C09082=1012.478,318.787,350.070,169.822,52.836,160.283
C09083=1012.472,318.539,350.102,169.815,52.841,160.283
C09084=1012.466,318.291,350.134,169.808,52.848,160.283
C09085=1012.460,318.044,350.167,169.801,52.853,160.283
C09086=1012.455,317.796,350.200,169.794,52.859,160.283
C09087=1012.449,317.549,350.233,169.787,52.865,160.283
C09088=1012.443,317.301,350.265,169.780,52.871,160.283
C09089=1012.436,317.053,350.298,169.774,52.876,160.283
C09090=1012.430,316.805,350.330,169.767,52.883,160.283
C09091=1012.424,316.557,350.362,169.760,52.889,160.283
C09092=1012.419,316.309,350.396,169.753,52.894,160.283
C09093=1012.412,316.062,350.429,169.746,52.900,160.283
C09094=1012.406,315.813,350.461,169.739,52.906,160.283
C09095=1012.400,315.566,350.493,169.732,52.912,160.283
C09096=1012.394,315.319,350.526,169.726,52.918,160.283
C09097=1012.388,315.071,350.558,169.719,52.924,160.283
C09098=1012.383,314.823,350.591,169.713,52.929,160.283
C09099=1012.377,314.575,350.623,169.705,52.936,160.283
C09100=1012.370,314.327,350.656,169.699,52.941,160.283
C09101=1012.365,314.080,350.687,169.692,52.948,160.283
C09102=1012.359,313.832,350.720,169.686,52.953,160.283
C09103=1012.353,313.583,350.753,169.678,52.959,160.283
C09104=1012.347,313.336,350.786,169.672,52.965,160.283
C09105=1012.342,313.088,350.817,169.665,52.971,160.283
C09106=1012.336,312.841,350.850,169.659,52.977,160.283
C09107=1012.330,312.593,350.882,169.652,52.983,160.283
C09108=1012.324,312.345,350.914,169.645,52.989,160.283
C09109=1012.319,312.097,350.947,169.638,52.995,160.283
C09110=1012.313,311.849,350.979,169.632,53.001,160.283
C09111=1012.307,311.602,351.011,169.625,53.007,160.283
C09112=1012.301,311.354,351.043,169.618,53.013,160.283
C09113=1012.295,311.106,351.075,169.611,53.019,160.283
C09114=1012.290,310.858,351.107,169.605,53.025,160.283
C09115=1012.284,310.610,351.140,169.598,53.032,160.283
C09116=1012.279,310.363,351.172,169.592,53.037,160.283
C09117=1012.273,310.114,351.204,169.585,53.044,160.283
C09118=1012.267,309.867,351.236,169.579,53.049,160.283
C09119=1012.261,309.619,351.269,169.572,53.056,160.283
C09120=1012.256,309.372,351.300,169.566,53.062,160.284
C09121=1012.250,309.123,351.333,169.558,53.068,160.283
C09122=1012.245,308.876,351.364,169.552,53.074,160.284
C09123=1012.237,308.577,351.403,169.544,53.082,160.284
C09124=1012.230,308.277,351.440,169.536,53.089,160.284
C09125=1012.222,307.977,351.479,169.528,53.097,160.284
C09126=1012.216,307.678,351.516,169.520,53.105,160.284
C09127=1012.209,307.431,351.548,169.514,53.111,160.284
C09128=1012.203,307.182,351.580,169.507,53.118,160.284
C09129=1012.198,306.935,351.610,169.500,53.124,160.284
C09130=1012.192,306.686,351.642,169.494,53.130,160.285
C09131=1012.186,306.439,351.673,169.487,53.136,160.285
C09132=1012.180,306.190,351.704,169.481,53.143,160.285
C09133=1012.174,305.943,351.735,169.474,53.149,160.285
C09134=1012.168,305.695,351.767,169.468,53.155,160.285
C09135=1012.162,305.447,351.798,169.461,53.162,160.285
C09136=1012.156,305.199,351.830,169.454,53.169,160.285
C09137=1012.150,304.951,351.860,169.448,53.175,160.286
C09138=1012.144,304.703,351.892,169.441,53.181,160.285
C09139=1012.138,304.455,351.923,169.435,53.188,160.286
C09140=1012.133,304.207,351.954,169.429,53.195,160.286
C09141=1012.127,303.959,351.985,169.422,53.200,160.286
C09142=1012.121,303.711,352.017,169.416,53.207,160.286
C09143=1012.115,303.464,352.047,169.410,53.214,160.287
C09144=1012.109,303.215,352.079,169.403,53.220,160.287
C09145=1012.104,302.968,352.109,169.396,53.227,160.287
C09146=1012.098,302.719,352.140,169.390,53.233,160.287
C09147=1012.092,302.471,352.172,169.384,53.240,160.287
C09148=1012.087,302.223,352.203,169.378,53.247,160.287
C09149=1012.082,301.975,352.234,169.371,53.253,160.287
C09150=1012.075,301.728,352.265,169.365,53.259,160.288
C09151=1012.070,301.479,352.296,169.358,53.266,160.288
C09152=1012.064,301.231,352.326,169.352,53.273,160.288
C09153=1012.059,300.984,352.358,169.346,53.279,160.288
C09154=1012.053,300.736,352.388,169.339,53.285,160.288
C09155=1012.047,300.487,352.420,169.333,53.292,160.289
C09156=1012.041,300.239,352.450,169.326,53.299,160.289
C09157=1012.036,299.992,352.482,169.320,53.305,160.289
C09158=1012.030,299.744,352.512,169.313,53.312,160.289
C09159=1012.025,299.496,352.543,169.308,53.319,160.289
C09160=1012.019,299.247,352.574,169.301,53.326,160.290
C09161=1012.013,298.999,352.605,169.295,53.332,160.290
C09162=1012.008,298.752,352.635,169.288,53.339,160.290
C09163=1012.002,298.504,352.667,169.283,53.346,160.290
C09164=1011.996,298.256,352.697,169.276,53.352,160.291
C09165=1011.991,298.008,352.728,169.270,53.359,160.291
C09166=1011.986,297.760,352.758,169.263,53.365,160.291
C09167=1011.980,297.512,352.789,169.257,53.373,160.291
C09168=1011.975,297.264,352.820,169.251,53.379,160.291
C09169=1011.969,297.015,352.851,169.244,53.386,160.292
C09170=1011.963,296.768,352.881,169.239,53.393,160.292
C09171=1011.958,296.519,352.912,169.232,53.400,160.292
C09172=1011.952,296.272,352.942,169.226,53.406,160.292
C09173=1011.947,296.024,352.973,169.219,53.413,160.293
C09174=1011.941,295.776,353.004,169.214,53.419,160.293
C09175=1011.936,295.528,353.035,169.207,53.426,160.293
C09176=1011.931,295.279,353.064,169.201,53.433,160.293
C09177=1011.926,295.031,353.095,169.194,53.440,160.293
C09178=1011.920,294.783,353.126,169.189,53.446,160.294
C09179=1011.914,294.503,353.161,169.181,53.454,160.294
C09180=1011.908,294.222,353.195,169.174,53.462,160.294
C09181=1011.903,293.941,353.229,169.168,53.470,160.295
C09182=1011.896,293.661,353.264,169.161,53.478,160.295
C09183=1011.891,293.412,353.294,169.155,53.484,160.295
C09184=1011.885,293.163,353.326,169.148,53.491,160.295
C09185=1011.880,292.915,353.355,169.142,53.499,160.296
C09186=1011.875,292.667,353.386,169.136,53.505,160.296
C09187=1011.870,292.418,353.416,169.129,53.512,160.296
C09188=1011.864,292.170,353.447,169.124,53.519,160.297
C09189=1011.858,291.922,353.477,169.117,53.526,160.297
C09190=1011.853,291.674,353.507,169.112,53.533,160.297
C09191=1011.848,291.427,353.537,169.105,53.540,160.298
C09192=1011.843,291.178,353.567,169.100,53.547,160.298
C09193=1011.837,290.929,353.597,169.093,53.554,160.298
C09194=1011.832,290.682,353.627,169.087,53.561,160.298
C09195=1011.826,290.433,353.657,169.081,53.568,160.299
C09196=1011.820,290.185,353.687,169.075,53.576,160.299
C09197=1011.815,289.938,353.716,169.069,53.582,160.299
C09198=1011.810,289.689,353.746,169.063,53.590,160.300
C09199=1011.804,289.441,353.776,169.057,53.596,160.300
C09200=1011.799,289.193,353.806,169.051,53.604,160.300
C09201=1011.793,288.944,353.835,169.044,53.611,160.301
C09202=1011.788,288.697,353.865,169.039,53.618,160.301
C09203=1011.782,288.449,353.895,169.032,53.625,160.301
C09204=1011.777,288.200,353.925,169.027,53.632,160.302
C09205=1011.771,287.952,353.954,169.021,53.640,160.302
C09206=1011.766,287.704,353.984,169.014,53.647,160.302
C09207=1011.761,287.456,354.013,169.009,53.654,160.303
C09208=1011.755,287.207,354.043,169.002,53.661,160.303
C09209=1011.750,286.960,354.073,168.997,53.668,160.304
C09210=1011.745,286.712,354.102,168.990,53.676,160.304
C09211=1011.739,286.463,354.132,168.984,53.683,160.304
C09212=1011.734,286.216,354.161,168.978,53.690,160.305
C09213=1011.729,285.967,354.191,168.972,53.698,160.305
C09214=1011.723,285.719,354.221,168.967,53.704,160.305
C09215=1011.718,285.471,354.250,168.960,53.712,160.306
C09216=1011.713,285.223,354.280,168.954,53.719,160.306
C09217=1011.707,284.974,354.309,168.949,53.727,160.307
C09218=1011.702,284.726,354.338,168.942,53.734,160.307
C09219=1011.697,284.460,354.369,168.936,53.742,160.307
C09220=1011.691,284.195,354.401,168.930,53.750,160.308
C09221=1011.685,283.929,354.432,168.924,53.757,160.308
C09222=1011.679,283.664,354.464,168.917,53.765,160.308
C09223=1011.451,285.193,353.918,168.925,53.799,160.318
C09224=1011.460,285.578,353.873,168.935,53.789,160.318
C09225=1011.468,285.963,353.827,168.945,53.777,160.317
C09226=1011.477,286.348,353.782,168.954,53.766,160.316
C09227=1011.484,286.732,353.736,168.962,53.754,160.316
C09228=1011.490,286.981,353.706,168.969,53.747,160.316
C09229=1011.495,287.229,353.677,168.975,53.740,160.315
C09230=1011.500,287.477,353.648,168.981,53.733,160.315
C09231=1011.506,287.725,353.618,168.987,53.726,160.315
C09232=1011.511,287.973,353.589,168.992,53.718,160.314
C09233=1011.516,288.221,353.558,168.999,53.711,160.314
C09234=1011.522,288.469,353.529,169.005,53.704,160.314
C09235=1011.527,288.718,353.499,169.011,53.697,160.313
C09236=1011.532,288.966,353.470,169.017,53.690,160.313
C09237=1011.538,289.214,353.440,169.024,53.682,160.313
C09238=1011.544,289.462,353.410,169.029,53.675,160.312
C09239=1011.549,289.710,353.380,169.036,53.668,160.312
C09240=1011.554,289.958,353.351,169.041,53.661,160.312
C09241=1011.560,290.207,353.321,169.048,53.654,160.311
C09242=1011.565,290.454,353.291,169.054,53.647,160.311
C09243=1011.570,290.703,353.261,169.060,53.640,160.311
C09244=1011.575,290.951,353.231,169.066,53.633,160.310
C09245=1011.581,291.199,353.201,169.072,53.626,160.310
C09246=1011.586,291.447,353.171,169.078,53.618,160.310
C09247=1011.592,291.695,353.141,169.085,53.611,160.310
C09248=1011.598,291.943,353.111,169.091,53.605,160.309
C09249=1011.603,292.190,353.081,169.097,53.597,160.309
C09250=1011.608,292.439,353.051,169.103,53.591,160.309
C09251=1011.614,292.687,353.021,169.109,53.584,160.308
C09252=1011.619,292.970,352.986,169.117,53.576,160.308
C09253=1011.625,293.254,352.952,169.123,53.568,160.308
C09254=1011.631,293.539,352.916,169.130,53.560,160.307
C09255=1011.638,293.822,352.882,169.137,53.552,160.307
C09256=1011.643,294.070,352.851,169.143,53.546,160.307
C09257=1011.648,294.317,352.822,169.150,53.539,160.307
C09258=1011.653,294.566,352.791,169.156,53.531,160.306
C09259=1011.659,294.813,352.760,169.162,53.525,160.306
C09260=1011.664,295.062,352.729,169.169,53.518,160.306
C09261=1011.670,295.309,352.699,169.174,53.511,160.306
C09262=1011.675,295.558,352.668,169.181,53.504,160.305
C09263=1011.679,295.806,352.638,169.187,53.498,160.305
C09264=1011.685,296.054,352.607,169.193,53.491,160.305
C09265=1011.690,296.302,352.577,169.199,53.484,160.305
C09266=1011.696,296.550,352.546,169.205,53.477,160.304
C09267=1011.701,296.798,352.515,169.212,53.470,160.304
C09268=1011.707,297.046,352.485,169.218,53.463,160.304
C09269=1011.712,297.294,352.454,169.225,53.457,160.304
C09270=1011.718,297.542,352.424,169.230,53.450,160.303
C09271=1011.723,297.790,352.393,169.237,53.443,160.303
C09272=1011.729,298.038,352.362,169.243,53.437,160.303
C09273=1011.734,298.286,352.331,169.249,53.430,160.303
C09274=1011.740,298.534,352.301,169.255,53.423,160.302
C09275=1011.745,298.782,352.270,169.262,53.416,160.302
C09276=1011.751,299.031,352.239,169.269,53.409,160.302
C09277=1011.756,299.279,352.208,169.275,53.404,160.302
C09278=1011.762,299.526,352.178,169.282,53.397,160.302
C09279=1011.767,299.775,352.147,169.287,53.390,160.302
C09280=1011.773,300.022,352.116,169.294,53.383,160.301
C09281=1011.778,300.270,352.085,169.300,53.377,160.301
C09282=1011.784,300.518,352.055,169.307,53.370,160.301
C09283=1011.790,300.767,352.023,169.313,53.363,160.301
C09284=1011.796,301.014,351.993,169.319,53.356,160.301
C09285=1011.801,301.262,351.961,169.326,53.350,160.301
C09286=1011.807,301.510,351.931,169.332,53.344,160.300
C09287=1011.812,301.758,351.900,169.339,53.337,160.300
C09288=1011.818,302.006,351.869,169.344,53.330,160.300
C09289=1011.824,302.254,351.838,169.351,53.324,160.300
C09290=1011.830,302.502,351.807,169.358,53.317,160.300
C09291=1011.835,302.750,351.776,169.364,53.311,160.299
C09292=1011.841,302.998,351.745,169.371,53.304,160.299
C09293=1011.846,303.246,351.714,169.377,53.297,160.299
C09294=1011.852,303.494,351.684,169.384,53.291,160.299
C09295=1011.858,303.742,351.652,169.391,53.284,160.299
C09296=1011.864,303.990,351.621,169.396,53.278,160.299
C09297=1011.869,304.237,351.590,169.404,53.272,160.299
C09298=1011.876,304.486,351.559,169.409,53.265,160.298
C09299=1011.881,304.734,351.528,169.416,53.258,160.298
C09300=1011.886,304.981,351.496,169.422,53.253,160.298
C09301=1011.893,305.230,351.466,169.429,53.246,160.298
C09302=1011.898,305.477,351.434,169.436,53.239,160.298
C09303=1011.905,305.725,351.403,169.442,53.233,160.298
C09304=1011.910,305.974,351.372,169.449,53.226,160.298
C09305=1011.916,306.221,351.341,169.455,53.220,160.297
C09306=1011.922,306.470,351.309,169.462,53.213,160.297
C09307=1011.928,306.717,351.278,169.469,53.207,160.297
C09308=1011.934,306.966,351.247,169.475,53.201,160.297
C09309=1011.940,307.213,351.216,169.482,53.195,160.297
C09310=1011.946,307.461,351.184,169.487,53.188,160.297
C09311=1011.952,307.709,351.153,169.495,53.182,160.297
C09312=1011.959,308.010,351.114,169.503,53.174,160.297
C09313=1011.966,308.312,351.077,169.511,53.166,160.297
C09314=1011.973,308.614,351.039,169.519,53.158,160.296
C09315=1011.980,308.915,351.000,169.527,53.151,160.296
C09316=1011.986,309.163,350.968,169.534,53.145,160.296
C09317=1011.992,309.411,350.936,169.540,53.139,160.296
C09318=1011.998,309.659,350.904,169.547,53.132,160.296
C09319=1012.003,309.906,350.872,169.553,53.126,160.296
C09320=1012.008,310.155,350.840,169.560,53.120,160.296
C09321=1012.014,310.402,350.808,169.567,53.114,160.296
C09322=1012.020,310.650,350.775,169.573,53.107,160.296
C09323=1012.026,310.898,350.743,169.580,53.102,160.296
C09324=1012.031,311.146,350.712,169.587,53.095,160.296
C09325=1012.037,311.394,350.680,169.593,53.090,160.296
C09326=1012.042,311.641,350.647,169.600,53.084,160.296
C09327=1012.048,311.889,350.615,169.606,53.078,160.296
C09328=1012.054,312.137,350.583,169.614,53.072,160.296
C09329=1012.060,312.384,350.550,169.620,53.066,160.296
C09330=1012.066,312.633,350.518,169.627,53.059,160.295
C09331=1012.071,312.880,350.486,169.633,53.053,160.295
C09332=1012.077,313.128,350.453,169.640,53.047,160.295
C09333=1012.083,313.376,350.421,169.647,53.041,160.295
C09334=1012.088,313.624,350.389,169.654,53.035,160.295
C09335=1012.094,313.871,350.357,169.661,53.029,160.295
C09336=1012.100,314.120,350.325,169.667,53.023,160.295
C09337=1012.107,314.367,350.292,169.674,53.017,160.295
C09338=1012.111,314.615,350.260,169.680,53.011,160.295
C09339=1012.118,314.863,350.227,169.688,53.005,160.295
C09340=1012.124,315.111,350.195,169.694,52.999,160.295
C09341=1012.130,315.358,350.162,169.701,52.993,160.295
C09342=1012.136,315.607,350.130,169.709,52.988,160.296
C09343=1012.142,315.854,350.098,169.715,52.982,160.296
C09344=1012.147,316.101,350.064,169.722,52.976,160.296
C09345=1012.153,316.350,350.032,169.728,52.970,160.295
C09346=1012.160,316.597,350.000,169.736,52.964,160.296
C09347=1012.165,316.845,349.968,169.742,52.958,160.295
C09348=1012.172,317.093,349.935,169.749,52.952,160.295
C09349=1012.177,317.340,349.903,169.757,52.946,160.296
C09350=1012.183,317.588,349.869,169.763,52.941,160.296
C09351=1012.189,317.836,349.837,169.770,52.934,160.296
C09352=1012.195,318.084,349.804,169.776,52.929,160.296
C09353=1012.202,318.331,349.772,169.784,52.923,160.296
C09354=1012.208,318.579,349.739,169.791,52.917,160.296
C09355=1012.213,318.827,349.706,169.797,52.911,160.296
C09356=1012.219,319.075,349.674,169.805,52.905,160.296
C09357=1012.226,319.323,349.641,169.811,52.900,160.296
C09358=1012.232,319.570,349.608,169.819,52.894,160.296
C09359=1012.238,319.818,349.575,169.826,52.888,160.296
C09360=1012.245,320.065,349.543,169.832,52.883,160.296
C09361=1012.250,320.314,349.510,169.840,52.877,160.296
C09362=1012.256,320.561,349.477,169.846,52.871,160.296
C09363=1012.262,320.809,349.444,169.854,52.865,160.296
C09364=1012.269,321.057,349.412,169.861,52.859,160.296
C09365=1012.276,321.305,349.379,169.867,52.854,160.297
C09366=1012.281,321.553,349.345,169.875,52.848,160.297
C09367=1012.287,321.800,349.313,169.881,52.843,160.297
C09368=1012.294,322.048,349.280,169.889,52.837,160.297
C09369=1012.300,322.296,349.247,169.896,52.831,160.297
C09370=1012.306,322.543,349.214,169.903,52.826,160.297
C09371=1012.312,322.791,349.181,169.910,52.820,160.297
C09372=1012.321,323.099,349.140,169.919,52.813,160.297
C09373=1012.328,323.406,349.099,169.927,52.806,160.297
C09374=1012.337,323.713,349.058,169.936,52.799,160.298
C09375=1012.344,324.020,349.017,169.945,52.792,160.298
C09376=1012.350,324.268,348.984,169.952,52.786,160.298
C09377=1012.357,324.515,348.950,169.960,52.781,160.298
C09378=1012.364,324.763,348.918,169.967,52.775,160.298
C09379=1012.369,325.011,348.884,169.973,52.770,160.298
C09380=1012.376,325.258,348.851,169.981,52.764,160.298
C09381=1012.383,325.506,348.818,169.988,52.758,160.298
C09382=1012.388,325.754,348.784,169.995,52.753,160.299
C09383=1012.395,326.001,348.751,170.003,52.748,160.299
C09384=1012.401,326.249,348.717,170.010,52.742,160.299
C09385=1012.407,326.497,348.683,170.017,52.737,160.299
C09386=1012.413,326.744,348.650,170.024,52.731,160.299
C09387=1012.420,326.992,348.616,170.031,52.726,160.299
C09388=1012.426,327.239,348.583,170.039,52.721,160.300
C09389=1012.432,327.487,348.549,170.046,52.715,160.300
C09390=1012.438,327.735,348.515,170.053,52.710,160.300
C09391=1012.445,327.982,348.481,170.061,52.705,160.300
C09392=1012.451,328.230,348.447,170.068,52.699,160.300
C09393=1012.457,328.478,348.413,170.075,52.694,160.301
C09394=1012.463,328.725,348.380,170.083,52.689,160.301
C09395=1012.470,328.973,348.346,170.089,52.684,160.301
C09396=1012.476,329.220,348.312,170.097,52.678,160.301
C09397=1012.483,329.468,348.278,170.105,52.673,160.301
C09398=1012.489,329.715,348.244,170.111,52.668,160.302
C09399=1012.495,329.963,348.209,170.119,52.662,160.302
C09400=1012.502,330.211,348.177,170.127,52.657,160.302
C09401=1012.508,330.459,348.142,170.133,52.652,160.302
C09402=1012.514,330.706,348.108,170.141,52.646,160.302
C09403=1012.521,330.954,348.074,170.149,52.641,160.303
C09404=1012.527,331.201,348.040,170.156,52.636,160.303
C09405=1012.534,331.449,348.006,170.164,52.631,160.303
C09406=1012.541,331.697,347.972,170.171,52.625,160.303
C09407=1012.546,331.944,347.938,170.178,52.620,160.304
C09408=1012.553,332.191,347.903,170.186,52.615,160.304
C09409=1012.559,332.439,347.869,170.194,52.610,160.304
C09410=1012.566,332.687,347.834,170.200,52.605,160.304
C09411=1012.573,332.934,347.801,170.208,52.600,160.305
C09412=1012.579,333.182,347.766,170.216,52.594,160.305
C09413=1012.585,333.429,347.731,170.223,52.590,160.305
C09414=1012.592,333.677,347.697,170.231,52.584,160.305
C09415=1012.598,333.924,347.663,170.238,52.580,160.306
C09416=1012.604,334.172,347.628,170.245,52.575,160.306
C09417=1012.611,334.420,347.593,170.253,52.569,160.306
C09418=1012.617,334.667,347.559,170.261,52.564,160.307
C09419=1012.624,334.914,347.524,170.268,52.559,160.307
C09420=1012.630,335.162,347.490,170.276,52.555,160.307
C09421=1012.637,335.410,347.455,170.284,52.549,160.308
C09422=1012.644,335.657,347.421,170.291,52.545,160.308
C09423=1012.650,335.904,347.386,170.298,52.539,160.308
C09424=1012.657,336.152,347.352,170.307,52.535,160.309
C09425=1012.663,336.399,347.316,170.313,52.530,160.309
C09426=1012.670,336.647,347.282,170.321,52.525,160.309
C09427=1012.677,336.895,347.247,170.329,52.519,160.309
C09428=1012.683,337.143,347.212,170.336,52.515,160.310
C09429=1012.689,337.389,347.178,170.344,52.510,160.310
C09430=1012.696,337.637,347.143,170.352,52.505,160.310
C09431=1012.702,337.885,347.108,170.360,52.500,160.311
C09432=1012.711,338.188,347.065,170.369,52.494,160.311
C09433=1012.719,338.491,347.022,170.378,52.488,160.312
C09434=1012.727,338.794,346.980,170.388,52.482,160.312
C09435=1012.736,339.096,346.936,170.397,52.477,160.313
C09436=1012.743,339.343,346.901,170.405,52.471,160.313
C09437=1012.748,339.592,346.866,170.413,52.466,160.313
C09438=1012.755,339.839,346.831,170.420,52.462,160.314
C09439=1012.762,340.086,346.796,170.428,52.457,160.314
C09440=1012.769,340.334,346.761,170.436,52.453,160.315
C09441=1012.775,340.581,346.726,170.445,52.448,160.315
C09442=1012.782,340.828,346.691,170.451,52.443,160.315
C09443=1012.788,341.076,346.655,170.459,52.438,160.316
C09444=1012.795,341.323,346.619,170.467,52.433,160.316
C09445=1012.802,341.570,346.584,170.476,52.428,160.317
C09446=1012.809,341.818,346.549,170.483,52.424,160.317
C09447=1012.815,342.065,346.514,170.491,52.419,160.317
C09448=1012.822,342.313,346.478,170.499,52.415,160.318
C09449=1012.829,342.561,346.442,170.507,52.410,160.318
C09450=1012.836,342.807,346.407,170.514,52.405,160.319
C09451=1012.843,343.055,346.371,170.522,52.401,160.319
C09452=1012.849,343.303,346.336,170.530,52.396,160.319
C09453=1012.856,343.549,346.300,170.539,52.392,160.320
C09454=1012.863,343.797,346.264,170.546,52.387,160.320
C09455=1012.870,344.045,346.229,170.554,52.383,160.321
C09456=1012.876,344.292,346.193,170.562,52.378,160.321
C09457=1012.883,344.539,346.158,170.571,52.373,160.322
C09458=1012.890,344.787,346.122,170.579,52.368,160.322
C09459=1012.898,345.034,346.086,170.586,52.365,160.323
C09460=1012.904,345.282,346.051,170.594,52.360,160.323
C09461=1012.911,345.528,346.015,170.602,52.355,160.324
C09462=1012.918,345.776,345.979,170.611,52.350,160.324
C09463=1012.925,346.023,345.943,170.619,52.346,160.325
C09464=1012.931,346.270,345.907,170.626,52.342,160.325
C09465=1012.939,346.518,345.871,170.634,52.337,160.326
C09466=1012.945,346.765,345.835,170.643,52.333,160.326
C09467=1012.953,347.013,345.799,170.651,52.328,160.327
C09468=1012.959,347.260,345.763,170.659,52.324,160.327
C09469=1012.966,347.507,345.727,170.667,52.320,160.328
C09470=1012.974,347.755,345.691,170.675,52.315,160.328
C09471=1012.980,348.002,345.654,170.683,52.311,160.329
C09472=1012.987,348.249,345.618,170.691,52.306,160.329
C09473=1012.994,348.496,345.582,170.700,52.302,160.330
C09474=1013.000,348.743,345.545,170.708,52.297,160.330
C09475=1013.008,348.991,345.509,170.716,52.294,160.331
C09476=1013.014,349.238,345.473,170.724,52.290,160.332
C09477=1013.022,349.485,345.437,170.732,52.285,160.332
C09478=1013.028,349.732,345.400,170.741,52.281,160.333
C09479=1013.036,349.980,345.364,170.749,52.276,160.333
C09480=1013.043,350.227,345.327,170.758,52.272,160.334
C09481=1013.050,350.474,345.291,170.766,52.268,160.334
C09482=1013.057,350.722,345.254,170.774,52.263,160.335
C09483=1013.064,350.969,345.219,170.782,52.259,160.335
C09484=1013.071,351.216,345.182,170.790,52.255,160.336
C09485=1013.079,351.464,345.145,170.799,52.251,160.337
C09486=1013.085,351.710,345.108,170.807,52.246,160.337
C09487=1013.093,351.958,345.072,170.816,52.242,160.338
C09488=1013.100,352.206,345.035,170.824,52.238,160.338
C09489=1013.107,352.452,344.999,170.833,52.234,160.339
C09490=1013.114,352.699,344.962,170.841,52.230,160.340
C09491=1013.122,352.947,344.926,170.850,52.226,160.340
C09492=1013.130,353.247,344.881,170.860,52.220,160.341
C09493=1013.139,353.547,344.837,170.869,52.216,160.342
C09494=1013.148,353.848,344.791,170.880,52.211,160.343
C09495=1013.156,354.148,344.747,170.890,52.206,160.343
C09496=1013.164,354.395,344.709,170.899,52.201,160.344
C09497=1013.171,354.643,344.673,170.908,52.198,160.345
C09498=1013.178,354.890,344.635,170.916,52.194,160.345
C09499=1013.185,355.136,344.598,170.925,52.190,160.346
C09500=1013.192,355.384,344.562,170.933,52.186,160.347
C09501=1013.199,355.631,344.524,170.942,52.182,160.347
C09502=1013.207,355.878,344.487,170.950,52.178,160.348
C09503=1013.214,356.125,344.450,170.959,52.173,160.349
C09504=1013.222,356.372,344.413,170.968,52.169,160.349
C09505=1013.229,356.620,344.375,170.977,52.166,160.350
C09506=1013.237,356.866,344.338,170.985,52.162,160.351
C09507=1013.244,357.114,344.301,170.994,52.158,160.351
C09508=1013.250,357.361,344.264,171.002,52.154,160.352
C09509=1013.258,357.608,344.227,171.011,52.150,160.353
C09510=1013.266,357.855,344.190,171.020,52.146,160.354
C09511=1013.273,358.102,344.152,171.028,52.142,160.354
C09512=1013.280,358.349,344.115,171.037,52.139,160.355
C09513=1013.288,358.597,344.077,171.046,52.134,160.356
C09514=1013.295,358.843,344.039,171.054,52.130,160.356
C09515=1013.303,359.090,344.001,171.063,52.127,160.357
C09516=1013.310,359.337,343.964,171.072,52.123,160.358
C09517=1013.317,359.585,343.926,171.081,52.119,160.359
C09518=1013.324,359.832,343.889,171.089,52.115,160.359
C09519=1013.332,360.078,343.850,171.098,52.112,160.360
C09520=1013.339,360.325,343.813,171.107,52.108,160.361
C09521=1013.346,360.573,343.775,171.116,52.104,160.362
C09522=1013.354,360.819,343.737,171.125,52.101,160.363
C09523=1013.361,361.066,343.700,171.133,52.097,160.363
C09524=1013.369,361.313,343.661,171.142,52.093,160.364
C09525=1013.377,361.561,343.623,171.151,52.090,160.365
C09526=1013.384,361.808,343.586,171.160,52.086,160.366
C09527=1013.391,362.054,343.548,171.169,52.082,160.367
C09528=1013.399,362.301,343.509,171.179,52.078,160.368
C09529=1013.407,362.549,343.472,171.188,52.075,160.368
C09530=1013.414,362.795,343.433,171.196,52.071,160.369
C09531=1013.422,363.042,343.396,171.205,52.067,160.370
C09532=1013.430,363.289,343.357,171.214,52.064,160.371
C09533=1013.437,363.536,343.319,171.223,52.061,160.372
C09534=1013.445,363.783,343.281,171.232,52.057,160.373
C09535=1013.453,364.030,343.243,171.241,52.054,160.373
C09536=1013.460,364.277,343.205,171.251,52.050,160.374
C09537=1013.467,364.524,343.166,171.260,52.046,160.375
C09538=1013.475,364.771,343.128,171.269,52.043,160.376
C09539=1013.482,365.018,343.090,171.278,52.039,160.377
C09540=1013.491,365.265,343.051,171.287,52.036,160.378
C09541=1013.498,365.512,343.013,171.296,52.033,160.379
C09542=1013.506,365.759,342.974,171.306,52.029,160.380
C09543=1013.514,366.005,342.936,171.315,52.025,160.380
C09544=1013.522,366.253,342.898,171.324,52.022,160.381
C09545=1013.529,366.500,342.860,171.333,52.018,160.382
C09546=1013.537,366.747,342.821,171.343,52.015,160.383
C09547=1013.545,366.993,342.782,171.352,52.011,160.384
C09548=1013.553,367.240,342.744,171.361,52.008,160.385
C09549=1013.560,367.487,342.705,171.370,52.005,160.386
C09550=1013.568,367.734,342.666,171.379,52.001,160.387
C09551=1013.576,367.980,342.627,171.389,51.998,160.388
C09552=1013.586,368.288,342.579,171.401,51.994,160.389
C09553=1013.596,368.596,342.530,171.413,51.989,160.390
C09554=1013.605,368.905,342.482,171.424,51.986,160.391
C09555=1013.615,369.212,342.433,171.436,51.981,160.393
C09556=1013.622,369.459,342.394,171.445,51.978,160.394
C09557=1013.631,369.706,342.354,171.454,51.975,160.394
C09558=1013.638,369.952,342.316,171.465,51.972,160.396
C09559=1013.646,370.199,342.276,171.474,51.968,160.397
C09560=1013.654,370.446,342.238,171.483,51.965,160.398
C09561=1013.663,370.693,342.198,171.493,51.962,160.399
C09562=1013.670,370.939,342.159,171.502,51.959,160.400
C09563=1013.678,371.187,342.120,171.512,51.956,160.401
C09564=1013.686,371.433,342.080,171.522,51.952,160.402
C09565=1013.694,371.680,342.041,171.531,51.949,160.403
C09566=1013.702,371.927,342.002,171.541,51.947,160.404
C09567=1013.710,372.174,341.962,171.551,51.943,160.405
C09568=1013.718,372.421,341.923,171.560,51.940,160.406
C09569=1013.726,372.667,341.884,171.569,51.937,160.407
C09570=1013.734,372.914,341.844,171.580,51.934,160.408
C09571=1013.742,373.160,341.805,171.589,51.930,160.409
C09572=1013.751,373.407,341.765,171.599,51.927,160.410
C09573=1013.759,373.654,341.726,171.609,51.924,160.411
C09574=1013.767,373.900,341.686,171.619,51.921,160.412
C09575=1013.775,374.147,341.647,171.628,51.918,160.413
C09576=1013.783,374.394,341.607,171.638,51.915,160.414
C09577=1013.792,374.640,341.568,171.648,51.912,160.416
C09578=1013.799,374.887,341.528,171.657,51.909,160.417
C09579=1013.808,375.134,341.488,171.668,51.906,160.418
C09580=1013.816,375.381,341.448,171.677,51.903,160.419
C09581=1013.825,375.627,341.408,171.688,51.900,160.420
C09582=1013.833,375.874,341.368,171.697,51.897,160.421
C09583=1013.840,376.121,341.328,171.707,51.894,160.422
C09584=1013.848,376.367,341.288,171.717,51.891,160.423
C09585=1013.857,376.614,341.248,171.728,51.889,160.425
C09586=1013.865,376.860,341.208,171.737,51.886,160.426
C09587=1013.873,377.107,341.168,171.747,51.883,160.427
C09588=1013.881,377.353,341.128,171.757,51.880,160.428
C09589=1013.890,377.601,341.087,171.768,51.877,160.429
C09590=1013.898,377.847,341.047,171.777,51.875,160.431
C09591=1013.906,378.093,341.007,171.787,51.871,160.432
C09592=1013.914,378.340,340.967,171.797,51.869,160.433
C09593=1013.923,378.587,340.926,171.808,51.866,160.434
C09594=1013.931,378.833,340.885,171.817,51.864,160.435
C09595=1013.940,379.079,340.845,171.828,51.860,160.437
C09596=1013.948,379.327,340.805,171.839,51.858,160.438
C09597=1013.956,379.573,340.764,171.848,51.855,160.439
C09598=1013.965,379.819,340.724,171.859,51.852,160.440
C09599=1013.973,380.066,340.683,171.869,51.849,160.442
C09600=1013.981,380.312,340.643,171.879,51.847,160.443
C09601=1013.991,380.559,340.602,171.889,51.844,160.444
C09602=1013.999,380.805,340.561,171.899,51.842,160.445
C09603=1014.007,381.052,340.521,171.910,51.839,160.447
C09604=1014.016,381.298,340.480,171.921,51.836,160.448
C09605=1014.024,381.545,340.440,171.930,51.834,160.449
C09606=1014.033,381.792,340.399,171.941,51.831,160.451
C09607=1014.041,382.039,340.358,171.952,51.828,160.452
C09608=1014.050,382.285,340.318,171.963,51.826,160.453
C09609=1014.059,382.532,340.277,171.972,51.823,160.454
C09610=1014.067,382.777,340.235,171.983,51.820,160.456
C09611=1014.076,383.024,340.195,171.994,51.818,160.457
C09612=1014.089,383.406,340.131,172.010,51.814,160.459
C09613=1014.103,383.787,340.068,172.026,51.810,160.461
C09614=1014.117,384.170,340.004,172.042,51.806,160.463
C09615=1014.130,384.552,339.940,172.060,51.802,160.466
C09616=1014.139,384.799,339.899,172.070,51.800,160.467
C09617=1014.148,385.044,339.859,172.080,51.798,160.468
C09618=1014.157,385.290,339.817,172.091,51.795,160.470
C09619=1014.166,385.537,339.776,172.102,51.792,160.471
C09620=1014.175,385.784,339.734,172.113,51.790,160.473
C09621=1014.183,386.030,339.693,172.124,51.788,160.474
C09622=1014.192,386.276,339.651,172.134,51.786,160.475
C09623=1014.201,386.522,339.610,172.145,51.783,160.477
C09624=1014.209,386.769,339.569,172.156,51.781,160.478
C09625=1014.218,387.015,339.527,172.167,51.778,160.480
C09626=1014.227,387.262,339.485,172.178,51.776,160.481
C09627=1014.236,387.508,339.443,172.189,51.774,160.483
C09628=1014.245,387.755,339.402,172.200,51.772,160.484
C09629=1014.254,388.001,339.360,172.211,51.769,160.486
C09630=1014.263,388.247,339.317,172.222,51.767,160.487
C09631=1014.272,388.493,339.276,172.233,51.765,160.489
C09632=1014.280,388.740,339.233,172.244,51.763,160.490
C09633=1014.289,388.986,339.192,172.255,51.761,160.492
C09634=1014.298,389.232,339.150,172.266,51.758,160.493
C09635=1014.307,389.478,339.108,172.277,51.756,160.495
C09636=1014.316,389.725,339.066,172.288,51.754,160.496
C09637=1014.325,389.971,339.024,172.299,51.751,160.498
C09638=1014.335,390.217,338.982,172.310,51.749,160.499
C09639=1014.344,390.463,338.940,172.322,51.747,160.501
C09640=1013.996,388.410,338.943,172.211,51.825,160.501
C09641=1013.987,388.163,338.985,172.200,51.828,160.499
C09642=1013.978,387.917,339.027,172.189,51.830,160.498
C09643=1013.969,387.671,339.068,172.178,51.833,160.496
C09644=1013.960,387.424,339.110,172.168,51.835,160.495
C09645=1013.952,387.179,339.151,172.157,51.837,160.493
C09646=1013.943,386.932,339.193,172.146,51.839,160.492
C09647=1013.934,386.686,339.235,172.135,51.841,160.490
C09648=1013.925,386.440,339.277,172.124,51.844,160.489
C09649=1013.916,386.193,339.318,172.113,51.847,160.488
C09650=1013.907,385.946,339.359,172.102,51.849,160.486
C09651=1013.899,385.701,339.401,172.091,51.851,160.485
C09652=1013.890,385.454,339.442,172.080,51.854,160.483
C09653=1013.881,385.207,339.483,172.070,51.856,160.482
C09654=1013.872,384.961,339.525,172.059,51.859,160.480
C09655=1013.864,384.715,339.566,172.049,51.861,160.479
C09656=1013.855,384.468,339.607,172.038,51.864,160.478
C09657=1013.843,384.127,339.664,172.023,51.867,160.476
C09658=1013.831,383.785,339.721,172.008,51.871,160.474
C09659=1013.819,383.443,339.778,171.993,51.874,160.472
C09660=1013.806,383.102,339.834,171.979,51.878,160.470
C09661=1013.798,382.855,339.875,171.968,51.881,160.469
C09662=1013.790,382.609,339.916,171.958,51.883,160.467
C09663=1013.780,382.362,339.956,171.947,51.886,160.466
C09664=1013.771,382.116,339.998,171.936,51.888,160.465
C09665=1013.763,381.869,340.039,171.926,51.892,160.464
C09666=1013.754,381.623,340.079,171.915,51.894,160.462
C09667=1013.746,381.376,340.120,171.905,51.896,160.461
C09668=1013.737,381.129,340.161,171.895,51.900,160.460
C09669=1013.729,380.883,340.201,171.884,51.902,160.458
C09670=1013.721,380.637,340.241,171.874,51.904,160.457
C09671=1013.712,380.390,340.282,171.864,51.908,160.456
C09672=1013.704,380.144,340.323,171.853,51.910,160.454
C09673=1013.695,379.897,340.363,171.844,51.913,160.453
C09674=1013.687,379.650,340.403,171.833,51.916,160.452
C09675=1013.679,379.404,340.444,171.823,51.919,160.451
C09676=1013.669,379.157,340.484,171.813,51.921,160.450
C09677=1013.661,378.911,340.525,171.802,51.924,160.448
C09678=1013.654,378.664,340.565,171.792,51.927,160.447
C09679=1013.644,378.417,340.605,171.782,51.930,160.446
C09680=1013.636,378.171,340.646,171.772,51.933,160.445
C09681=1013.629,377.924,340.686,171.761,51.936,160.443
C09682=1013.620,377.678,340.726,171.752,51.938,160.442
C09683=1013.612,377.431,340.766,171.741,51.942,160.441
C09684=1013.603,377.184,340.807,171.731,51.944,160.440
C09685=1013.596,376.937,340.847,171.721,51.947,160.439
C09686=1013.587,376.691,340.887,171.712,51.950,160.438
C09687=1013.579,376.445,340.927,171.701,51.953,160.436
C09688=1013.571,376.198,340.967,171.692,51.956,160.435
C09689=1013.563,375.952,341.007,171.682,51.959,160.434
C09690=1013.555,375.705,341.047,171.672,51.961,160.433
C09691=1013.547,375.459,341.087,171.661,51.965,160.432
C09692=1013.539,375.212,341.127,171.652,51.967,160.431
C09693=1013.531,374.965,341.166,171.642,51.971,160.429
C09694=1013.522,374.718,341.206,171.632,51.973,160.428
C09695=1013.515,374.472,341.246,171.622,51.977,160.427
C09696=1013.506,374.225,341.285,171.613,51.980,160.426
C09697=1013.498,373.978,341.324,171.602,51.983,160.425
C09698=1013.490,373.731,341.364,171.593,51.986,160.424
C09699=1013.482,373.485,341.404,171.583,51.989,160.423
C09700=1013.473,373.238,341.443,171.573,51.992,160.422
C09701=1013.465,372.991,341.483,171.563,51.995,160.421
C09702=1013.457,372.745,341.522,171.554,51.999,160.420
C09703=1013.449,372.498,341.562,171.543,52.002,160.419
C09704=1013.441,372.251,341.601,171.534,52.005,160.418
C09705=1013.433,372.004,341.640,171.524,52.009,160.417
C09706=1013.425,371.757,341.680,171.515,52.012,160.416
C09707=1013.417,371.511,341.719,171.505,52.014,160.414
C09708=1013.409,371.264,341.757,171.495,52.018,160.414
C09709=1013.401,371.017,341.797,171.486,52.021,160.412
C09710=1013.393,370.770,341.836,171.476,52.025,160.412
C09711=1013.385,370.524,341.875,171.467,52.028,160.410
C09712=1013.377,370.277,341.915,171.457,52.031,160.409
C09713=1013.369,370.030,341.953,171.447,52.034,160.408
C09714=1013.361,369.783,341.993,171.438,52.038,160.408
C09715=1013.354,369.536,342.032,171.429,52.041,160.406
C09716=1013.346,369.290,342.071,171.419,52.045,160.405
C09717=1013.336,368.979,342.120,171.408,52.048,160.404
C09718=1013.327,368.669,342.168,171.396,52.053,160.403
C09719=1013.316,368.359,342.218,171.383,52.057,160.402
C09720=1013.307,368.049,342.267,171.372,52.061,160.401
C09721=1013.299,367.802,342.305,171.362,52.065,160.400
C09722=1013.291,367.556,342.344,171.353,52.068,160.399
C09723=1013.284,367.308,342.383,171.344,52.071,160.398
C09724=1013.276,367.062,342.422,171.335,52.075,160.397
C09725=1013.268,366.814,342.460,171.325,52.078,160.396
C09726=1013.261,366.568,342.499,171.316,52.082,160.395
C09727=1013.252,366.321,342.537,171.307,52.085,160.394
C09728=1013.245,366.074,342.575,171.298,52.088,160.393
C09729=1013.237,365.827,342.614,171.288,52.092,160.392
C09730=1013.229,365.580,342.652,171.279,52.096,160.391
C09731=1013.221,365.333,342.691,171.270,52.099,160.390
C09732=1013.215,365.086,342.729,171.261,52.102,160.390
C09733=1013.207,364.839,342.767,171.251,52.106,160.389
C09734=1013.199,364.592,342.806,171.242,52.110,160.388
C09735=1013.191,364.346,342.844,171.233,52.114,160.387
C09736=1013.183,364.098,342.882,171.224,52.117,160.386
C09737=1013.176,363.851,342.920,171.215,52.121,160.385
C09738=1013.168,363.605,342.958,171.205,52.125,160.384
C09739=1013.161,363.357,342.996,171.196,52.128,160.383
C09740=1013.153,363.110,343.035,171.187,52.132,160.383
C09741=1013.145,362.864,343.073,171.179,52.136,160.382
C09742=1013.138,362.617,343.110,171.170,52.139,160.381
C09743=1013.130,362.369,343.149,171.160,52.143,160.380
C09744=1013.123,362.122,343.186,171.151,52.146,160.379
C09745=1013.115,361.876,343.225,171.142,52.150,160.379
C09746=1013.108,361.629,343.262,171.133,52.154,160.378
C09747=1013.101,361.382,343.300,171.124,52.157,160.377
C09748=1013.093,361.134,343.338,171.116,52.161,160.376
C09749=1013.085,360.887,343.376,171.107,52.165,160.375
C09750=1013.078,360.640,343.413,171.098,52.169,160.375
C09751=1013.071,360.394,343.452,171.089,52.173,160.374
C09752=1013.063,360.146,343.489,171.080,52.177,160.373
C09753=1013.056,359.899,343.527,171.071,52.180,160.372
C09754=1013.049,359.653,343.565,171.062,52.185,160.372
C09755=1013.041,359.406,343.602,171.053,52.188,160.371
C09756=1013.034,359.158,343.640,171.045,52.192,160.370
C09757=1013.027,358.911,343.678,171.036,52.196,160.369
C09758=1013.020,358.664,343.715,171.027,52.200,160.369
C09759=1013.012,358.417,343.753,171.018,52.203,160.368
C09760=1013.005,358.170,343.790,171.010,52.207,160.367
C09761=1012.998,357.923,343.828,171.001,52.211,160.366
C09762=1012.990,357.676,343.865,170.992,52.215,160.365
C09763=1012.983,357.429,343.902,170.984,52.219,160.365
C09764=1012.975,357.182,343.940,170.975,52.223,160.364
C09765=1012.968,356.935,343.977,170.966,52.227,160.364
C09766=1012.961,356.687,344.015,170.958,52.231,160.363
C09767=1012.953,356.440,344.051,170.949,52.235,160.362
C09768=1012.946,356.193,344.088,170.940,52.239,160.361
C09769=1012.939,355.946,344.126,170.931,52.243,160.361
C09770=1012.932,355.699,344.162,170.922,52.247,160.360
C09771=1012.924,355.452,344.199,170.914,52.251,160.359
C09772=1012.917,355.205,344.237,170.905,52.256,160.359
C09773=1012.910,354.957,344.274,170.897,52.260,160.358
C09774=1012.902,354.710,344.311,170.888,52.264,160.357
C09775=1012.896,354.463,344.347,170.880,52.268,160.357
C09776=1012.889,354.216,344.385,170.871,52.272,160.356
C09777=1012.880,353.913,344.430,170.861,52.276,160.355
C09778=1012.872,353.611,344.475,170.851,52.281,160.354
C09779=1012.862,353.308,344.519,170.841,52.287,160.354
C09780=1012.853,353.005,344.565,170.830,52.292,160.353
C09781=1012.846,352.759,344.602,170.822,52.296,160.352
C09782=1012.839,352.511,344.638,170.813,52.300,160.352
C09783=1012.832,352.264,344.675,170.805,52.304,160.351
C09784=1012.825,352.017,344.711,170.796,52.309,160.351
C09785=1012.817,351.770,344.748,170.788,52.313,160.350
C09786=1012.810,351.522,344.784,170.779,52.317,160.349
C09787=1012.803,351.275,344.821,170.771,52.321,160.349
C09788=1012.797,351.028,344.858,170.763,52.326,160.348
C09789=1012.789,350.781,344.893,170.754,52.330,160.347
C09790=1012.783,350.533,344.930,170.746,52.334,160.347
C09791=1012.775,350.286,344.966,170.737,52.339,160.346
C09792=1012.769,350.039,345.003,170.729,52.343,160.346
C09793=1012.761,349.791,345.039,170.721,52.348,160.345
C09794=1012.754,349.544,345.076,170.712,52.352,160.345
C09795=1012.747,349.297,345.112,170.705,52.356,160.344
C09796=1012.740,349.050,345.148,170.697,52.360,160.344
C09797=1012.733,348.802,345.184,170.688,52.364,160.343
C09798=1012.726,348.555,345.221,170.680,52.369,160.342
C09799=1012.719,348.308,345.257,170.671,52.373,160.342
C09800=1012.712,348.061,345.294,170.663,52.378,160.341
C09801=1012.705,347.814,345.329,170.655,52.382,160.341
C09802=1012.699,347.565,345.365,170.647,52.387,160.340
C09803=1012.692,347.319,345.401,170.639,52.391,160.340
C09804=1012.685,347.072,345.438,170.631,52.395,160.339
C09805=1012.678,346.824,345.473,170.623,52.400,160.339
C09806=1012.671,346.577,345.509,170.614,52.404,160.338
C09807=1012.665,346.330,345.546,170.606,52.409,160.338
C09808=1012.657,346.082,345.581,170.598,52.414,160.337
C09809=1012.651,345.835,345.618,170.589,52.418,160.337
C09810=1012.644,345.587,345.653,170.582,52.422,160.336
C09811=1012.637,345.340,345.689,170.574,52.427,160.336
C09812=1012.630,345.092,345.724,170.566,52.432,160.335
C09813=1012.623,344.845,345.760,170.558,52.437,160.335
C09814=1012.617,344.598,345.796,170.549,52.441,160.334
C09815=1012.609,344.351,345.831,170.541,52.446,160.334
C09816=1012.602,344.103,345.867,170.534,52.450,160.333
C09817=1012.596,343.856,345.903,170.526,52.455,160.333
C09818=1012.589,343.609,345.939,170.518,52.459,160.333
C09819=1012.582,343.361,345.974,170.510,52.464,160.332
C09820=1012.575,343.114,346.009,170.502,52.469,160.332
C09821=1012.569,342.866,346.045,170.495,52.473,160.331
C09822=1012.562,342.619,346.081,170.487,52.478,160.331
C09823=1012.555,342.372,346.116,170.478,52.483,160.330
C09824=1012.548,342.124,346.151,170.470,52.488,160.330
C09825=1012.542,341.877,346.187,170.462,52.492,160.329
C09826=1012.535,341.629,346.222,170.455,52.497,160.329
C09827=1012.529,341.382,346.257,170.447,52.502,160.329
C09828=1012.522,341.134,346.292,170.439,52.506,160.328
C09829=1012.515,340.887,346.327,170.431,52.511,160.328
C09830=1012.508,340.640,346.362,170.423,52.516,160.327
C09831=1012.502,340.392,346.398,170.415,52.520,160.327
C09832=1012.496,340.145,346.433,170.408,52.526,160.327
C09833=1012.489,339.897,346.468,170.400,52.531,160.326
C09834=1012.482,339.650,346.504,170.392,52.535,160.326
C09835=1012.475,339.403,346.539,170.384,52.540,160.325
C09836=1012.468,339.155,346.574,170.376,52.545,160.325
C09837=1012.460,338.850,346.617,170.367,52.551,160.325
C09838=1012.453,338.545,346.661,170.357,52.557,160.324
C09839=1012.445,338.239,346.703,170.347,52.563,160.324
C09840=1012.437,337.934,346.747,170.339,52.569,160.323
C09841=1012.430,337.686,346.782,170.330,52.574,160.323
C09842=1012.423,337.439,346.815,170.323,52.579,160.323
C09843=1012.416,337.192,346.850,170.315,52.584,160.322
C09844=1012.410,336.945,346.886,170.308,52.588,160.322
C09845=1012.403,336.697,346.920,170.300,52.594,160.322
C09846=1012.396,336.449,346.955,170.292,52.599,160.321
C09847=1012.390,336.201,346.990,170.284,52.604,160.321
C09848=1012.384,335.955,347.024,170.277,52.608,160.321
C09849=1012.377,335.707,347.059,170.269,52.614,160.320
C09850=1012.371,335.459,347.093,170.261,52.619,160.320
C09851=1012.364,335.211,347.128,170.253,52.624,160.320
C09852=1012.358,334.964,347.162,170.246,52.628,160.319
C09853=1012.351,334.717,347.197,170.239,52.634,160.319
C09854=1012.344,334.469,347.231,170.231,52.639,160.319
C09855=1012.338,334.221,347.266,170.224,52.644,160.318
C09856=1012.332,333.974,347.301,170.216,52.649,160.318
C09857=1012.325,333.726,347.335,170.209,52.655,160.318
C09858=1012.319,333.478,347.369,170.200,52.659,160.318
C09859=1012.313,333.231,347.403,170.194,52.665,160.317
C09860=1012.306,332.984,347.439,170.186,52.670,160.317
C09861=1012.300,332.736,347.473,170.178,52.675,160.317
C09862=1012.294,332.488,347.507,170.171,52.680,160.317
C09863=1012.287,332.241,347.541,170.164,52.685,160.316
C09864=1012.281,331.993,347.575,170.156,52.691,160.316
C09865=1012.274,331.745,347.609,170.149,52.695,160.316
C09866=1012.268,331.498,347.643,170.141,52.701,160.315
C09867=1012.261,331.250,347.677,170.133,52.706,160.315
C09868=1012.255,331.003,347.711,170.127,52.711,160.315
C09869=1012.249,330.755,347.746,170.119,52.717,160.315
C09870=1012.242,330.508,347.779,170.111,52.722,160.315
C09871=1012.236,330.260,347.814,170.104,52.727,160.314
C09872=1012.230,330.013,347.848,170.097,52.733,160.314
C09873=1012.223,329.765,347.881,170.089,52.738,160.314
C09874=1012.217,329.517,347.915,170.082,52.743,160.314
C09875=1012.211,329.269,347.949,170.075,52.749,160.314
C09876=1012.204,329.022,347.983,170.067,52.754,160.313
C09877=1012.198,328.774,348.017,170.060,52.759,160.313
C09878=1012.192,328.527,348.050,170.053,52.765,160.313
C09879=1012.186,328.280,348.084,170.045,52.770,160.313
C09880=1012.179,328.032,348.118,170.038,52.775,160.313
C09881=1012.172,327.785,348.152,170.031,52.781,160.312
C09882=1012.166,327.536,348.185,170.023,52.786,160.312
C09883=1012.160,327.289,348.220,170.016,52.791,160.312
C09884=1012.154,327.041,348.252,170.009,52.797,160.312
C09885=1012.148,326.793,348.287,170.001,52.802,160.311
C09886=1012.142,326.546,348.321,169.994,52.807,160.311
C09887=1012.136,326.298,348.353,169.987,52.813,160.311
C09888=1012.130,326.051,348.388,169.980,52.819,160.311
C09889=1012.124,325.802,348.421,169.973,52.824,160.311
C09890=1012.117,325.555,348.455,169.965,52.829,160.311
C09891=1012.111,325.307,348.488,169.958,52.835,160.311
C09892=1012.105,325.060,348.521,169.952,52.840,160.310
C09893=1012.098,324.812,348.555,169.944,52.846,160.310
C09894=1012.092,324.565,348.587,169.937,52.852,160.310
C09895=1012.085,324.317,348.620,169.929,52.858,160.310
C09896=1012.080,324.069,348.653,169.922,52.863,160.310
C09897=1012.071,323.759,348.695,169.914,52.870,160.310
C09898=1012.063,323.450,348.736,169.904,52.877,160.310
C09899=1012.056,323.140,348.777,169.895,52.884,160.309
C09900=1012.047,322.831,348.818,169.886,52.892,160.309
C09901=1012.041,322.583,348.851,169.880,52.897,160.309
C09902=1012.036,322.336,348.884,169.872,52.903,160.309
C09903=1012.029,322.088,348.917,169.865,52.908,160.309
C09904=1012.023,321.840,348.950,169.859,52.914,160.309
C09905=1012.016,321.592,348.983,169.851,52.920,160.309
C09906=1012.010,321.345,349.016,169.844,52.926,160.309
C09907=1012.004,321.097,349.049,169.837,52.931,160.309
C09908=1011.998,320.849,349.082,169.830,52.937,160.309
C09909=1011.992,320.601,349.114,169.823,52.943,160.309
C09910=1011.985,320.354,349.147,169.816,52.948,160.308
C09911=1011.979,320.106,349.179,169.809,52.954,160.308
C09912=1011.973,319.858,349.212,169.802,52.959,160.308
C09913=1011.967,319.610,349.245,169.795,52.966,160.308
C09914=1011.961,319.363,349.278,169.788,52.972,160.308
C09915=1011.955,319.115,349.311,169.781,52.978,160.308
C09916=1011.949,318.867,349.343,169.774,52.983,160.308
C09917=1011.943,318.619,349.376,169.766,52.989,160.308
C09918=1011.937,318.371,349.409,169.760,52.995,160.308
C09919=1011.931,318.124,349.442,169.753,53.000,160.308
C09920=1011.925,317.876,349.473,169.746,53.006,160.308
C09921=1011.919,317.629,349.506,169.739,53.012,160.308
C09922=1011.913,317.381,349.539,169.732,53.019,160.308
C09923=1011.907,317.133,349.571,169.726,53.024,160.308
C09924=1011.901,316.885,349.604,169.718,53.030,160.307
C09925=1011.895,316.637,349.636,169.711,53.036,160.307
C09926=1011.889,316.389,349.669,169.705,53.042,160.308
C09927=1011.883,316.142,349.701,169.697,53.048,160.307
C09928=1011.877,315.894,349.733,169.691,53.054,160.308
C09929=1011.871,315.646,349.766,169.684,53.060,160.308
C09930=1011.866,315.398,349.799,169.677,53.066,160.307
C09931=1011.860,315.151,349.831,169.671,53.072,160.308
C09932=1011.854,314.903,349.863,169.663,53.078,160.308
C09933=1011.848,314.655,349.896,169.657,53.084,160.308
C09934=1011.842,314.407,349.928,169.650,53.090,160.308
C09935=1011.837,314.159,349.960,169.643,53.096,160.308
C09936=1011.831,313.911,349.993,169.637,53.102,160.308
C09937=1011.825,313.663,350.025,169.629,53.108,160.308
C09938=1011.819,313.416,350.057,169.623,53.114,160.308
C09939=1011.813,313.168,350.089,169.616,53.120,160.308
C09940=1011.807,312.920,350.121,169.610,53.126,160.308
C09941=1011.802,312.673,350.154,169.603,53.132,160.308
C09942=1011.796,312.425,350.186,169.595,53.138,160.308
C09943=1011.790,312.176,350.218,169.589,53.144,160.308
C09944=1011.785,311.929,350.250,169.582,53.150,160.308
C09945=1011.779,311.681,350.283,169.576,53.156,160.308
C09946=1011.773,311.434,350.314,169.568,53.162,160.308
C09947=1011.768,311.185,350.347,169.562,53.168,160.308
C09948=1011.763,310.938,350.379,169.556,53.175,160.308
C09949=1011.756,310.690,350.411,169.549,53.181,160.308
C09950=1011.751,310.443,350.443,169.542,53.187,160.308
C09951=1011.745,310.194,350.475,169.535,53.193,160.308
C09952=1011.740,309.947,350.507,169.529,53.199,160.308
C09953=1011.734,309.699,350.539,169.522,53.206,160.308
C09954=1011.729,309.451,350.571,169.516,53.211,160.308
C09955=1011.723,309.203,350.603,169.509,53.218,160.308
C09956=1011.718,308.955,350.635,169.502,53.223,160.308
C09957=1011.711,308.651,350.674,169.494,53.232,160.308
C09958=1011.703,308.347,350.712,169.486,53.239,160.308
C09959=1011.695,308.043,350.751,169.478,53.247,160.309
C09960=1011.688,307.740,350.789,169.469,53.255,160.309
C09961=1011.683,307.491,350.821,169.464,53.261,160.309
C09962=1011.677,307.244,350.852,169.456,53.268,160.309
C09963=1011.671,306.995,350.883,169.450,53.274,160.309
C09964=1011.665,306.748,350.914,169.443,53.280,160.309
C09965=1011.660,306.500,350.945,169.437,53.287,160.309
C09966=1011.653,306.252,350.976,169.430,53.293,160.309
C09967=1011.648,306.004,351.008,169.424,53.300,160.309
C09968=1011.641,305.756,351.039,169.416,53.306,160.309
C09969=1011.636,305.508,351.070,169.411,53.313,160.310
C09970=1011.630,305.260,351.101,169.404,53.319,160.310
C09971=1011.624,305.012,351.132,169.397,53.326,160.310
C09972=1011.618,304.764,351.163,169.391,53.332,160.310
C09973=1011.613,304.516,351.194,169.384,53.338,160.310
C09974=1011.606,304.268,351.225,169.378,53.345,160.310
C09975=1011.601,304.020,351.256,169.371,53.352,160.311
C09976=1011.595,303.772,351.287,169.364,53.358,160.310
C09977=1011.589,303.524,351.319,169.358,53.364,160.311
C09978=1011.584,303.276,351.349,169.352,53.371,160.311
C09979=1011.579,303.028,351.380,169.346,53.377,160.311
C09980=1011.572,302.781,351.411,169.339,53.384,160.311
C09981=1011.567,302.532,351.442,169.332,53.391,160.311
C09982=1011.561,302.284,351.473,169.326,53.397,160.312
C09983=1011.556,302.037,351.505,169.319,53.404,160.312
C09984=1011.550,301.789,351.535,169.313,53.410,160.312
C09985=1011.545,301.541,351.566,169.307,53.417,160.312
C09986=1011.538,301.292,351.597,169.300,53.424,160.312
C09987=1011.533,301.044,351.627,169.294,53.430,160.312
C09988=1011.527,300.797,351.659,169.287,53.437,160.312
C09989=1011.522,300.549,351.689,169.281,53.443,160.313
C09990=1011.517,300.301,351.720,169.275,53.450,160.313
C09991=1011.511,300.053,351.751,169.268,53.457,160.313
C09992=1011.506,299.805,351.782,169.262,53.464,160.313
C09993=1011.500,299.556,351.812,169.255,53.470,160.313
C09994=1011.494,299.308,351.843,169.250,53.477,160.314
C09995=1011.489,299.060,351.874,169.243,53.484,160.314
C09996=1011.484,298.812,351.905,169.236,53.491,160.314
//INST
///DATE 2021/06/25 14:50
///ATTR SC,RW,RJ
////FRAME ROBOT
///GROUP1 RB1
NOP
MOVL C00000 V=800.0 PL=0
MOVL C00001 V=800.0 PL=0
MOVL C00002 V=800.0 PL=0
MOVL C00003 V=800.0 PL=0
MOVL C00004 V=800.0 PL=0
MOVL C00005 V=800.0 PL=0
MOVL C00006 V=800.0 PL=0
MOVL C00007 V=800.0 PL=0
MOVL C00008 V=800.0 PL=0
MOVL C00009 V=800.0 PL=0
MOVL C00010 V=800.0 PL=0
MOVL C00011 V=800.0 PL=0
MOVL C00012 V=800.0 PL=0
MOVL C00013 V=800.0 PL=0
MOVL C00014 V=800.0 PL=0
MOVL C00015 V=800.0 PL=0
MOVL C00016 V=800.0 PL=0
MOVL C00017 V=800.0 PL=0
MOVL C00018 V=800.0 PL=0
MOVL C00019 V=800.0 PL=0
MOVL C00020 V=800.0 PL=0
MOVL C00021 V=800.0 PL=0
MOVL C00022 V=800.0 PL=0
MOVL C00023 V=800.0 PL=0
MOVL C00024 V=800.0 PL=0
MOVL C00025 V=800.0 PL=0
MOVL C00026 V=800.0 PL=0
MOVL C00027 V=800.0 PL=0
MOVL C00028 V=800.0 PL=0
MOVL C00029 V=800.0 PL=0
MOVL C00030 V=800.0 PL=0
MOVL C00031 V=800.0 PL=0
MOVL C00032 V=800.0 PL=0
MOVL C00033 V=800.0 PL=0
MOVL C00034 V=800.0 PL=0
MOVL C00035 V=800.0 PL=0
MOVL C00036 V=800.0 PL=0
MOVL C00037 V=800.0 PL=0
MOVL C00038 V=800.0 PL=0
MOVL C00039 V=800.0 PL=0
MOVL C00040 V=800.0 PL=0
MOVL C00041 V=800.0 PL=0
MOVL C00042 V=800.0 PL=0
MOVL C00043 V=800.0 PL=0
MOVL C00044 V=800.0 PL=0
MOVL C00045 V=800.0 PL=0
MOVL C00046 V=800.0 PL=0
MOVL C00047 V=800.0 PL=0
MOVL C00048 V=800.0 PL=0
MOVL C00049 V=800.0 PL=0
MOVL C00050 V=800.0 PL=0
MOVL C00051 V=800.0 PL=0
MOVL C00052 V=800.0 PL=0
MOVL C00053 V=800.0 PL=0
MOVL C00054 V=800.0 PL=0
MOVL C00055 V=800.0 PL=0
MOVL C00056 V=800.0 PL=0
MOVL C00057 V=800.0 PL=0
MOVL C00058 V=800.0 PL=0
MOVL C00059 V=800.0 PL=0
MOVL C00060 V=800.0 PL=0
MOVL C00061 V=800.0 PL=0
MOVL C00062 V=800.0 PL=0
MOVL C00063 V=800.0 PL=0
MOVL C00064 V=800.0 PL=0
MOVL C00065 V=800.0 PL=0
MOVL C00066 V=800.0 PL=0
MOVL C00067 V=800.0 PL=0
MOVL C00068 V=800.0 PL=0
MOVL C00069 V=800.0 PL=0
MOVL C00070 V=800.0 PL=0
MOVL C00071 V=800.0 PL=0
MOVL C00072 V=800.0 PL=0
MOVL C00073 V=800.0 PL=0
MOVL C00074 V=800.0 PL=0
MOVL C00075 V=800.0 PL=0
MOVL C00076 V=800.0 PL=0
MOVL C00077 V=800.0 PL=0
MOVL C00078 V=800.0 PL=0
MOVL C00079 V=800.0 PL=0
MOVL C00080 V=800.0 PL=0
MOVL C00081 V=800.0 PL=0
MOVL C00082 V=800.0 PL=0
MOVL C00083 V=800.0 PL=0
MOVL C00084 V=800.0 PL=0
MOVL C00085 V=800.0 PL=0
MOVL C00086 V=800.0 PL=0
MOVL C00087 V=800.0 PL=0
MOVL C00088 V=800.0 PL=0
MOVL C00089 V=800.0 PL=0
MOVL C00090 V=800.0 PL=0
MOVL C00091 V=800.0 PL=0
MOVL C00092 V=800.0 PL=0
MOVL C00093 V=800.0 PL=0
MOVL C00094 V=800.0 PL=0
MOVL C00095 V=800.0 PL=0
MOVL C00096 V=800.0 PL=0
MOVL C00097 V=800.0 PL=0
MOVL C00098 V=800.0 PL=0
MOVL C00099 V=800.0 PL=0
MOVL C00100 V=800.0 PL=0
MOVL C00101 V=800.0 PL=0
MOVL C00102 V=800.0 PL=0
MOVL C00103 V=800.0 PL=0
MOVL C00104 V=800.0 PL=0
MOVL C00105 V=800.0 PL=0
MOVL C00106 V=800.0 PL=0
MOVL C00107 V=800.0 PL=0
MOVL C00108 V=800.0 PL=0
MOVL C00109 V=800.0 PL=0
MOVL C00110 V=800.0 PL=0
MOVL C00111 V=800.0 PL=0
MOVL C00112 V=800.0 PL=0
MOVL C00113 V=800.0 PL=0
MOVL C00114 V=800.0 PL=0
MOVL C00115 V=800.0 PL=0
MOVL C00116 V=800.0 PL=0
MOVL C00117 V=800.0 PL=0
MOVL C00118 V=800.0 PL=0
MOVL C00119 V=800.0 PL=0
MOVL C00120 V=800.0 PL=0
MOVL C00121 V=800.0 PL=0
MOVL C00122 V=800.0 PL=0
MOVL C00123 V=800.0 PL=0
MOVL C00124 V=800.0 PL=0
MOVL C00125 V=800.0 PL=0
MOVL C00126 V=800.0 PL=0
MOVL C00127 V=800.0 PL=0
MOVL C00128 V=800.0 PL=0
MOVL C00129 V=800.0 PL=0
MOVL C00130 V=800.0 PL=0
MOVL C00131 V=800.0 PL=0
MOVL C00132 V=800.0 PL=0
MOVL C00133 V=800.0 PL=0
MOVL C00134 V=800.0 PL=0
MOVL C00135 V=800.0 PL=0
MOVL C00136 V=800.0 PL=0
MOVL C00137 V=800.0 PL=0
MOVL C00138 V=800.0 PL=0
MOVL C00139 V=800.0 PL=0
MOVL C00140 V=800.0 PL=0
MOVL C00141 V=800.0 PL=0
MOVL C00142 V=800.0 PL=0
MOVL C00143 V=800.0 PL=0
MOVL C00144 V=800.0 PL=0
MOVL C00145 V=800.0 PL=0
MOVL C00146 V=800.0 PL=0
MOVL C00147 V=800.0 PL=0
MOVL C00148 V=800.0 PL=0
MOVL C00149 V=800.0 PL=0
MOVL C00150 V=800.0 PL=0
MOVL C00151 V=800.0 PL=0
MOVL C00152 V=800.0 PL=0
MOVL C00153 V=800.0 PL=0
MOVL C00154 V=800.0 PL=0
MOVL C00155 V=800.0 PL=0
MOVL C00156 V=800.0 PL=0
MOVL C00157 V=800.0 PL=0
MOVL C00158 V=800.0 PL=0
MOVL C00159 V=800.0 PL=0
MOVL C00160 V=800.0 PL=0
MOVL C00161 V=800.0 PL=0
MOVL C00162 V=800.0 PL=0
MOVL C00163 V=800.0 PL=0
MOVL C00164 V=800.0 PL=0
MOVL C00165 V=800.0 PL=0
MOVL C00166 V=800.0 PL=0
MOVL C00167 V=800.0 PL=0
MOVL C00168 V=800.0 PL=0
MOVL C00169 V=800.0 PL=0
MOVL C00170 V=800.0 PL=0
MOVL C00171 V=800.0 PL=0
MOVL C00172 V=800.0 PL=0
MOVL C00173 V=800.0 PL=0
MOVL C00174 V=800.0 PL=0
MOVL C00175 V=800.0 PL=0
MOVL C00176 V=800.0 PL=0
MOVL C00177 V=800.0 PL=0
MOVL C00178 V=800.0 PL=0
MOVL C00179 V=800.0 PL=0
MOVL C00180 V=800.0 PL=0
MOVL C00181 V=800.0 PL=0
MOVL C00182 V=800.0 PL=0
MOVL C00183 V=800.0 PL=0
MOVL C00184 V=800.0 PL=0
MOVL C00185 V=800.0 PL=0
MOVL C00186 V=800.0 PL=0
MOVL C00187 V=800.0 PL=0
MOVL C00188 V=800.0 PL=0
MOVL C00189 V=800.0 PL=0
MOVL C00190 V=800.0 PL=0
MOVL C00191 V=800.0 PL=0
MOVL C00192 V=800.0 PL=0
MOVL C00193 V=800.0 PL=0
MOVL C00194 V=800.0 PL=0
MOVL C00195 V=800.0 PL=0
MOVL C00196 V=800.0 PL=0
MOVL C00197 V=800.0 PL=0
MOVL C00198 V=800.0 PL=0
MOVL C00199 V=800.0 PL=0
MOVL C00200 V=800.0 PL=0
MOVL C00201 V=800.0 PL=0
MOVL C00202 V=800.0 PL=0
MOVL C00203 V=800.0 PL=0
MOVL C00204 V=800.0 PL=0
MOVL C00205 V=800.0 PL=0
MOVL C00206 V=800.0 PL=0
MOVL C00207 V=800.0 PL=0
MOVL C00208 V=800.0 PL=0
MOVL C00209 V=800.0 PL=0
MOVL C00210 V=800.0 PL=0
MOVL C00211 V=800.0 PL=0
MOVL C00212 V=800.0 PL=0
MOVL C00213 V=800.0 PL=0
MOVL C00214 V=800.0 PL=0
MOVL C00215 V=800.0 PL=0
MOVL C00216 V=800.0 PL=0
MOVL C00217 V=800.0 PL=0
MOVL C00218 V=800.0 PL=0
MOVL C00219 V=800.0 PL=0
MOVL C00220 V=800.0 PL=0
MOVL C00221 V=800.0 PL=0
MOVL C00222 V=800.0 PL=0
MOVL C00223 V=800.0 PL=0
MOVL C00224 V=800.0 PL=0
MOVL C00225 V=800.0 PL=0
MOVL C00226 V=800.0 PL=0
MOVL C00227 V=800.0 PL=0
MOVL C00228 V=800.0 PL=0
MOVL C00229 V=800.0 PL=0
MOVL C00230 V=800.0 PL=0
MOVL C00231 V=800.0 PL=0
MOVL C00232 V=800.0 PL=0
MOVL C00233 V=800.0 PL=0
MOVL C00234 V=800.0 PL=0
MOVL C00235 V=800.0 PL=0
MOVL C00236 V=800.0 PL=0
MOVL C00237 V=800.0 PL=0
MOVL C00238 V=800.0 PL=0
MOVL C00239 V=800.0 PL=0
MOVL C00240 V=800.0 PL=0
MOVL C00241 V=800.0 PL=0
MOVL C00242 V=800.0 PL=0
MOVL C00243 V=800.0 PL=0
MOVL C00244 V=800.0 PL=0
MOVL C00245 V=800.0 PL=0
MOVL C00246 V=800.0 PL=0
MOVL C00247 V=800.0 PL=0
MOVL C00248 V=800.0 PL=0
MOVL C00249 V=800.0 PL=0
MOVL C00250 V=800.0 PL=0
MOVL C00251 V=800.0 PL=0
MOVL C00252 V=800.0 PL=0
MOVL C00253 V=800.0 PL=0
MOVL C00254 V=800.0 PL=0
MOVL C00255 V=800.0 PL=0
MOVL C00256 V=800.0 PL=0
MOVL C00257 V=800.0 PL=0
MOVL C00258 V=800.0 PL=0
MOVL C00259 V=800.0 PL=0
MOVL C00260 V=800.0 PL=0
MOVL C00261 V=800.0 PL=0
MOVL C00262 V=800.0 PL=0
MOVL C00263 V=800.0 PL=0
MOVL C00264 V=800.0 PL=0
MOVL C00265 V=800.0 PL=0
MOVL C00266 V=800.0 PL=0
MOVL C00267 V=800.0 PL=0
MOVL C00268 V=800.0 PL=0
MOVL C00269 V=800.0 PL=0
MOVL C00270 V=800.0 PL=0
MOVL C00271 V=800.0 PL=0
MOVL C00272 V=800.0 PL=0
MOVL C00273 V=800.0 PL=0
MOVL C00274 V=800.0 PL=0
MOVL C00275 V=800.0 PL=0
MOVL C00276 V=800.0 PL=0
MOVL C00277 V=800.0 PL=0
MOVL C00278 V=800.0 PL=0
MOVL C00279 V=800.0 PL=0
MOVL C00280 V=800.0 PL=0
MOVL C00281 V=800.0 PL=0
MOVL C00282 V=800.0 PL=0
MOVL C00283 V=800.0 PL=0
MOVL C00284 V=800.0 PL=0
MOVL C00285 V=800.0 PL=0
MOVL C00286 V=800.0 PL=0
MOVL C00287 V=800.0 PL=0
MOVL C00288 V=800.0 PL=0
MOVL C00289 V=800.0 PL=0
MOVL C00290 V=800.0 PL=0
MOVL C00291 V=800.0 PL=0
MOVL C00292 V=800.0 PL=0
MOVL C00293 V=800.0 PL=0
MOVL C00294 V=800.0 PL=0
MOVL C00295 V=800.0 PL=0
MOVL C00296 V=800.0 PL=0
MOVL C00297 V=800.0 PL=0
MOVL C00298 V=800.0 PL=0
MOVL C00299 V=800.0 PL=0
MOVL C00300 V=800.0 PL=0
MOVL C00301 V=800.0 PL=0
MOVL C00302 V=800.0 PL=0
MOVL C00303 V=800.0 PL=0
MOVL C00304 V=800.0 PL=0
MOVL C00305 V=800.0 PL=0
MOVL C00306 V=800.0 PL=0
MOVL C00307 V=800.0 PL=0
MOVL C00308 V=800.0 PL=0
MOVL C00309 V=800.0 PL=0
MOVL C00310 V=800.0 PL=0
MOVL C00311 V=800.0 PL=0
MOVL C00312 V=800.0 PL=0
MOVL C00313 V=800.0 PL=0
MOVL C00314 V=800.0 PL=0
MOVL C00315 V=800.0 PL=0
MOVL C00316 V=800.0 PL=0
MOVL C00317 V=800.0 PL=0
MOVL C00318 V=800.0 PL=0
MOVL C00319 V=800.0 PL=0
MOVL C00320 V=800.0 PL=0
MOVL C00321 V=800.0 PL=0
MOVL C00322 V=800.0 PL=0
MOVL C00323 V=800.0 PL=0
MOVL C00324 V=800.0 PL=0
MOVL C00325 V=800.0 PL=0
MOVL C00326 V=800.0 PL=0
MOVL C00327 V=800.0 PL=0
MOVL C00328 V=800.0 PL=0
MOVL C00329 V=800.0 PL=0
MOVL C00330 V=800.0 PL=0
MOVL C00331 V=800.0 PL=0
MOVL C00332 V=800.0 PL=0
MOVL C00333 V=800.0 PL=0
MOVL C00334 V=800.0 PL=0
MOVL C00335 V=800.0 PL=0
MOVL C00336 V=800.0 PL=0
MOVL C00337 V=800.0 PL=0
MOVL C00338 V=800.0 PL=0
MOVL C00339 V=800.0 PL=0
MOVL C00340 V=800.0 PL=0
MOVL C00341 V=800.0 PL=0
MOVL C00342 V=800.0 PL=0
MOVL C00343 V=800.0 PL=0
MOVL C00344 V=800.0 PL=0
MOVL C00345 V=800.0 PL=0
MOVL C00346 V=800.0 PL=0
MOVL C00347 V=800.0 PL=0
MOVL C00348 V=800.0 PL=0
MOVL C00349 V=800.0 PL=0
MOVL C00350 V=800.0 PL=0
MOVL C00351 V=800.0 PL=0
MOVL C00352 V=800.0 PL=0
MOVL C00353 V=800.0 PL=0
MOVL C00354 V=800.0 PL=0
MOVL C00355 V=800.0 PL=0
MOVL C00356 V=800.0 PL=0
MOVL C00357 V=800.0 PL=0
MOVL C00358 V=800.0 PL=0
MOVL C00359 V=800.0 PL=0
MOVL C00360 V=800.0 PL=0
MOVL C00361 V=800.0 PL=0
MOVL C00362 V=800.0 PL=0
MOVL C00363 V=800.0 PL=0
MOVL C00364 V=800.0 PL=0
MOVL C00365 V=800.0 PL=0
MOVL C00366 V=800.0 PL=0
MOVL C00367 V=800.0 PL=0
MOVL C00368 V=800.0 PL=0
MOVL C00369 V=800.0 PL=0
MOVL C00370 V=800.0 PL=0
MOVL C00371 V=800.0 PL=0
MOVL C00372 V=800.0 PL=0
MOVL C00373 V=800.0 PL=0
MOVL C00374 V=800.0 PL=0
MOVL C00375 V=800.0 PL=0
MOVL C00376 V=800.0 PL=0
MOVL C00377 V=800.0 PL=0
MOVL C00378 V=800.0 PL=0
MOVL C00379 V=800.0 PL=0
MOVL C00380 V=800.0 PL=0
MOVL C00381 V=800.0 PL=0
MOVL C00382 V=800.0 PL=0
MOVL C00383 V=800.0 PL=0
MOVL C00384 V=800.0 PL=0
MOVL C00385 V=800.0 PL=0
MOVL C00386 V=800.0 PL=0
MOVL C00387 V=800.0 PL=0
MOVL C00388 V=800.0 PL=0
MOVL C00389 V=800.0 PL=0
MOVL C00390 V=800.0 PL=0
MOVL C00391 V=800.0 PL=0
MOVL C00392 V=800.0 PL=0
MOVL C00393 V=800.0 PL=0
MOVL C00394 V=800.0 PL=0
MOVL C00395 V=800.0 PL=0
MOVL C00396 V=800.0 PL=0
MOVL C00397 V=800.0 PL=0
MOVL C00398 V=800.0 PL=0
MOVL C00399 V=800.0 PL=0
MOVL C00400 V=800.0 PL=0
MOVL C00401 V=800.0 PL=0
MOVL C00402 V=800.0 PL=0
MOVL C00403 V=800.0 PL=0
MOVL C00404 V=800.0 PL=0
MOVL C00405 V=800.0 PL=0
MOVL C00406 V=800.0 PL=0
MOVL C00407 V=800.0 PL=0
MOVL C00408 V=800.0 PL=0
MOVL C00409 V=800.0 PL=0
MOVL C00410 V=800.0 PL=0
MOVL C00411 V=800.0 PL=0
MOVL C00412 V=800.0 PL=0
MOVL C00413 V=800.0 PL=0
MOVL C00414 V=800.0 PL=0
MOVL C00415 V=800.0 PL=0
MOVL C00416 V=800.0 PL=0
MOVL C00417 V=800.0 PL=0
MOVL C00418 V=800.0 PL=0
MOVL C00419 V=800.0 PL=0
MOVL C00420 V=800.0 PL=0
MOVL C00421 V=800.0 PL=0
MOVL C00422 V=800.0 PL=0
MOVL C00423 V=800.0 PL=0
MOVL C00424 V=800.0 PL=0
MOVL C00425 V=800.0 PL=0
MOVL C00426 V=800.0 PL=0
MOVL C00427 V=800.0 PL=0
MOVL C00428 V=800.0 PL=0
MOVL C00429 V=800.0 PL=0
MOVL C00430 V=800.0 PL=0
MOVL C00431 V=800.0 PL=0
MOVL C00432 V=800.0 PL=0
MOVL C00433 V=800.0 PL=0
MOVL C00434 V=800.0 PL=0
MOVL C00435 V=800.0 PL=0
MOVL C00436 V=800.0 PL=0
MOVL C00437 V=800.0 PL=0
MOVL C00438 V=800.0 PL=0
MOVL C00439 V=800.0 PL=0
MOVL C00440 V=800.0 PL=0
MOVL C00441 V=800.0 PL=0
MOVL C00442 V=800.0 PL=0
MOVL C00443 V=800.0 PL=0
MOVL C00444 V=800.0 PL=0
MOVL C00445 V=800.0 PL=0
MOVL C00446 V=800.0 PL=0
MOVL C00447 V=800.0 PL=0
MOVL C00448 V=800.0 PL=0
MOVL C00449 V=800.0 PL=0
MOVL C00450 V=800.0 PL=0
MOVL C00451 V=800.0 PL=0
MOVL C00452 V=800.0 PL=0
MOVL C00453 V=800.0 PL=0
MOVL C00454 V=800.0 PL=0
MOVL C00455 V=800.0 PL=0
MOVL C00456 V=800.0 PL=0
MOVL C00457 V=800.0 PL=0
MOVL C00458 V=800.0 PL=0
MOVL C00459 V=800.0 PL=0
MOVL C00460 V=800.0 PL=0
MOVL C00461 V=800.0 PL=0
MOVL C00462 V=800.0 PL=0
MOVL C00463 V=800.0 PL=0
MOVL C00464 V=800.0 PL=0
MOVL C00465 V=800.0 PL=0
MOVL C00466 V=800.0 PL=0
MOVL C00467 V=800.0 PL=0
MOVL C00468 V=800.0 PL=0
MOVL C00469 V=800.0 PL=0
MOVL C00470 V=800.0 PL=0
MOVL C00471 V=800.0 PL=0
MOVL C00472 V=800.0 PL=0
MOVL C00473 V=800.0 PL=0
MOVL C00474 V=800.0 PL=0
MOVL C00475 V=800.0 PL=0
MOVL C00476 V=800.0 PL=0
MOVL C00477 V=800.0 PL=0
MOVL C00478 V=800.0 PL=0
MOVL C00479 V=800.0 PL=0
MOVL C00480 V=800.0 PL=0
MOVL C00481 V=800.0 PL=0
MOVL C00482 V=800.0 PL=0
MOVL C00483 V=800.0 PL=0
MOVL C00484 V=800.0 PL=0
MOVL C00485 V=800.0 PL=0
MOVL C00486 V=800.0 PL=0
MOVL C00487 V=800.0 PL=0
MOVL C00488 V=800.0 PL=0
MOVL C00489 V=800.0 PL=0
MOVL C00490 V=800.0 PL=0
MOVL C00491 V=800.0 PL=0
MOVL C00492 V=800.0 PL=0
MOVL C00493 V=800.0 PL=0
MOVL C00494 V=800.0 PL=0
MOVL C00495 V=800.0 PL=0
MOVL C00496 V=800.0 PL=0
MOVL C00497 V=800.0 PL=0
MOVL C00498 V=800.0 PL=0
MOVL C00499 V=800.0 PL=0
MOVL C00500 V=800.0 PL=0
MOVL C00501 V=800.0 PL=0
MOVL C00502 V=800.0 PL=0
MOVL C00503 V=800.0 PL=0
MOVL C00504 V=800.0 PL=0
MOVL C00505 V=800.0 PL=0
MOVL C00506 V=800.0 PL=0
MOVL C00507 V=800.0 PL=0
MOVL C00508 V=800.0 PL=0
MOVL C00509 V=800.0 PL=0
MOVL C00510 V=800.0 PL=0
MOVL C00511 V=800.0 PL=0
MOVL C00512 V=800.0 PL=0
MOVL C00513 V=800.0 PL=0
MOVL C00514 V=800.0 PL=0
MOVL C00515 V=800.0 PL=0
MOVL C00516 V=800.0 PL=0
MOVL C00517 V=800.0 PL=0
MOVL C00518 V=800.0 PL=0
MOVL C00519 V=800.0 PL=0
MOVL C00520 V=800.0 PL=0
MOVL C00521 V=800.0 PL=0
MOVL C00522 V=800.0 PL=0
MOVL C00523 V=800.0 PL=0
MOVL C00524 V=800.0 PL=0
MOVL C00525 V=800.0 PL=0
MOVL C00526 V=800.0 PL=0
MOVL C00527 V=800.0 PL=0
MOVL C00528 V=800.0 PL=0
MOVL C00529 V=800.0 PL=0
MOVL C00530 V=800.0 PL=0
MOVL C00531 V=800.0 PL=0
MOVL C00532 V=800.0 PL=0
MOVL C00533 V=800.0 PL=0
MOVL C00534 V=800.0 PL=0
MOVL C00535 V=800.0 PL=0
MOVL C00536 V=800.0 PL=0
MOVL C00537 V=800.0 PL=0
MOVL C00538 V=800.0 PL=0
MOVL C00539 V=800.0 PL=0
MOVL C00540 V=800.0 PL=0
MOVL C00541 V=800.0 PL=0
MOVL C00542 V=800.0 PL=0
MOVL C00543 V=800.0 PL=0
MOVL C00544 V=800.0 PL=0
MOVL C00545 V=800.0 PL=0
MOVL C00546 V=800.0 PL=0
MOVL C00547 V=800.0 PL=0
MOVL C00548 V=800.0 PL=0
MOVL C00549 V=800.0 PL=0
MOVL C00550 V=800.0 PL=0
MOVL C00551 V=800.0 PL=0
MOVL C00552 V=800.0 PL=0
MOVL C00553 V=800.0 PL=0
MOVL C00554 V=800.0 PL=0
MOVL C00555 V=800.0 PL=0
MOVL C00556 V=800.0 PL=0
MOVL C00557 V=800.0 PL=0
MOVL C00558 V=800.0 PL=0
MOVL C00559 V=800.0 PL=0
MOVL C00560 V=800.0 PL=0
MOVL C00561 V=800.0 PL=0
MOVL C00562 V=800.0 PL=0
MOVL C00563 V=800.0 PL=0
MOVL C00564 V=800.0 PL=0
MOVL C00565 V=800.0 PL=0
MOVL C00566 V=800.0 PL=0
MOVL C00567 V=800.0 PL=0
MOVL C00568 V=800.0 PL=0
MOVL C00569 V=800.0 PL=0
MOVL C00570 V=800.0 PL=0
MOVL C00571 V=800.0 PL=0
MOVL C00572 V=800.0 PL=0
MOVL C00573 V=800.0 PL=0
MOVL C00574 V=800.0 PL=0
MOVL C00575 V=800.0 PL=0
MOVL C00576 V=800.0 PL=0
MOVL C00577 V=800.0 PL=0
MOVL C00578 V=800.0 PL=0
MOVL C00579 V=800.0 PL=0
MOVL C00580 V=800.0 PL=0
MOVL C00581 V=800.0 PL=0
MOVL C00582 V=800.0 PL=0
MOVL C00583 V=800.0 PL=0
MOVL C00584 V=800.0 PL=0
MOVL C00585 V=800.0 PL=0
MOVL C00586 V=800.0 PL=0
MOVL C00587 V=800.0 PL=0
MOVL C00588 V=800.0 PL=0
MOVL C00589 V=800.0 PL=0
MOVL C00590 V=800.0 PL=0
MOVL C00591 V=800.0 PL=0
MOVL C00592 V=800.0 PL=0
MOVL C00593 V=800.0 PL=0
MOVL C00594 V=800.0 PL=0
MOVL C00595 V=800.0 PL=0
MOVL C00596 V=800.0 PL=0
MOVL C00597 V=800.0 PL=0
MOVL C00598 V=800.0 PL=0
MOVL C00599 V=800.0 PL=0
MOVL C00600 V=800.0 PL=0
MOVL C00601 V=800.0 PL=0
MOVL C00602 V=800.0 PL=0
MOVL C00603 V=800.0 PL=0
MOVL C00604 V=800.0 PL=0
MOVL C00605 V=800.0 PL=0
MOVL C00606 V=800.0 PL=0
MOVL C00607 V=800.0 PL=0
MOVL C00608 V=800.0 PL=0
MOVL C00609 V=800.0 PL=0
MOVL C00610 V=800.0 PL=0
MOVL C00611 V=800.0 PL=0
MOVL C00612 V=800.0 PL=0
MOVL C00613 V=800.0 PL=0
MOVL C00614 V=800.0 PL=0
MOVL C00615 V=800.0 PL=0
MOVL C00616 V=800.0 PL=0
MOVL C00617 V=800.0 PL=0
MOVL C00618 V=800.0 PL=0
MOVL C00619 V=800.0 PL=0
MOVL C00620 V=800.0 PL=0
MOVL C00621 V=800.0 PL=0
MOVL C00622 V=800.0 PL=0
MOVL C00623 V=800.0 PL=0
MOVL C00624 V=800.0 PL=0
MOVL C00625 V=800.0 PL=0
MOVL C00626 V=800.0 PL=0
MOVL C00627 V=800.0 PL=0
MOVL C00628 V=800.0 PL=0
MOVL C00629 V=800.0 PL=0
MOVL C00630 V=800.0 PL=0
MOVL C00631 V=800.0 PL=0
MOVL C00632 V=800.0 PL=0
MOVL C00633 V=800.0 PL=0
MOVL C00634 V=800.0 PL=0
MOVL C00635 V=800.0 PL=0
MOVL C00636 V=800.0 PL=0
MOVL C00637 V=800.0 PL=0
MOVL C00638 V=800.0 PL=0
MOVL C00639 V=800.0 PL=0
MOVL C00640 V=800.0 PL=0
MOVL C00641 V=800.0 PL=0
MOVL C00642 V=800.0 PL=0
MOVL C00643 V=800.0 PL=0
MOVL C00644 V=800.0 PL=0
MOVL C00645 V=800.0 PL=0
MOVL C00646 V=800.0 PL=0
MOVL C00647 V=800.0 PL=0
MOVL C00648 V=800.0 PL=0
MOVL C00649 V=800.0 PL=0
MOVL C00650 V=800.0 PL=0
MOVL C00651 V=800.0 PL=0
MOVL C00652 V=800.0 PL=0
MOVL C00653 V=800.0 PL=0
MOVL C00654 V=800.0 PL=0
MOVL C00655 V=800.0 PL=0
MOVL C00656 V=800.0 PL=0
MOVL C00657 V=800.0 PL=0
MOVL C00658 V=800.0 PL=0
MOVL C00659 V=800.0 PL=0
MOVL C00660 V=800.0 PL=0
MOVL C00661 V=800.0 PL=0
MOVL C00662 V=800.0 PL=0
MOVL C00663 V=800.0 PL=0
MOVL C00664 V=800.0 PL=0
MOVL C00665 V=800.0 PL=0
MOVL C00666 V=800.0 PL=0
MOVL C00667 V=800.0 PL=0
MOVL C00668 V=800.0 PL=0
MOVL C00669 V=800.0 PL=0
MOVL C00670 V=800.0 PL=0
MOVL C00671 V=800.0 PL=0
MOVL C00672 V=800.0 PL=0
MOVL C00673 V=800.0 PL=0
MOVL C00674 V=800.0 PL=0
MOVL C00675 V=800.0 PL=0
MOVL C00676 V=800.0 PL=0
MOVL C00677 V=800.0 PL=0
MOVL C00678 V=800.0 PL=0
MOVL C00679 V=800.0 PL=0
MOVL C00680 V=800.0 PL=0
MOVL C00681 V=800.0 PL=0
MOVL C00682 V=800.0 PL=0
MOVL C00683 V=800.0 PL=0
MOVL C00684 V=800.0 PL=0
MOVL C00685 V=800.0 PL=0
MOVL C00686 V=800.0 PL=0
MOVL C00687 V=800.0 PL=0
MOVL C00688 V=800.0 PL=0
MOVL C00689 V=800.0 PL=0
MOVL C00690 V=800.0 PL=0
MOVL C00691 V=800.0 PL=0
MOVL C00692 V=800.0 PL=0
MOVL C00693 V=800.0 PL=0
MOVL C00694 V=800.0 PL=0
MOVL C00695 V=800.0 PL=0
MOVL C00696 V=800.0 PL=0
MOVL C00697 V=800.0 PL=0
MOVL C00698 V=800.0 PL=0
MOVL C00699 V=800.0 PL=0
MOVL C00700 V=800.0 PL=0
MOVL C00701 V=800.0 PL=0
MOVL C00702 V=800.0 PL=0
MOVL C00703 V=800.0 PL=0
MOVL C00704 V=800.0 PL=0
MOVL C00705 V=800.0 PL=0
MOVL C00706 V=800.0 PL=0
MOVL C00707 V=800.0 PL=0
MOVL C00708 V=800.0 PL=0
MOVL C00709 V=800.0 PL=0
MOVL C00710 V=800.0 PL=0
MOVL C00711 V=800.0 PL=0
MOVL C00712 V=800.0 PL=0
MOVL C00713 V=800.0 PL=0
MOVL C00714 V=800.0 PL=0
MOVL C00715 V=800.0 PL=0
MOVL C00716 V=800.0 PL=0
MOVL C00717 V=800.0 PL=0
MOVL C00718 V=800.0 PL=0
MOVL C00719 V=800.0 PL=0
MOVL C00720 V=800.0 PL=0
MOVL C00721 V=800.0 PL=0
MOVL C00722 V=800.0 PL=0
MOVL C00723 V=800.0 PL=0
MOVL C00724 V=800.0 PL=0
MOVL C00725 V=800.0 PL=0
MOVL C00726 V=800.0 PL=0
MOVL C00727 V=800.0 PL=0
MOVL C00728 V=800.0 PL=0
MOVL C00729 V=800.0 PL=0
MOVL C00730 V=800.0 PL=0
MOVL C00731 V=800.0 PL=0
MOVL C00732 V=800.0 PL=0
MOVL C00733 V=800.0 PL=0
MOVL C00734 V=800.0 PL=0
MOVL C00735 V=800.0 PL=0
MOVL C00736 V=800.0 PL=0
MOVL C00737 V=800.0 PL=0
MOVL C00738 V=800.0 PL=0
MOVL C00739 V=800.0 PL=0
MOVL C00740 V=800.0 PL=0
MOVL C00741 V=800.0 PL=0
MOVL C00742 V=800.0 PL=0
MOVL C00743 V=800.0 PL=0
MOVL C00744 V=800.0 PL=0
MOVL C00745 V=800.0 PL=0
MOVL C00746 V=800.0 PL=0
MOVL C00747 V=800.0 PL=0
MOVL C00748 V=800.0 PL=0
MOVL C00749 V=800.0 PL=0
MOVL C00750 V=800.0 PL=0
MOVL C00751 V=800.0 PL=0
MOVL C00752 V=800.0 PL=0
MOVL C00753 V=800.0 PL=0
MOVL C00754 V=800.0 PL=0
MOVL C00755 V=800.0 PL=0
MOVL C00756 V=800.0 PL=0
MOVL C00757 V=800.0 PL=0
MOVL C00758 V=800.0 PL=0
MOVL C00759 V=800.0 PL=0
MOVL C00760 V=800.0 PL=0
MOVL C00761 V=800.0 PL=0
MOVL C00762 V=800.0 PL=0
MOVL C00763 V=800.0 PL=0
MOVL C00764 V=800.0 PL=0
MOVL C00765 V=800.0 PL=0
MOVL C00766 V=800.0 PL=0
MOVL C00767 V=800.0 PL=0
MOVL C00768 V=800.0 PL=0
MOVL C00769 V=800.0 PL=0
MOVL C00770 V=800.0 PL=0
MOVL C00771 V=800.0 PL=0
MOVL C00772 V=800.0 PL=0
MOVL C00773 V=800.0 PL=0
MOVL C00774 V=800.0 PL=0
MOVL C00775 V=800.0 PL=0
MOVL C00776 V=800.0 PL=0
MOVL C00777 V=800.0 PL=0
MOVL C00778 V=800.0 PL=0
MOVL C00779 V=800.0 PL=0
MOVL C00780 V=800.0 PL=0
MOVL C00781 V=800.0 PL=0
MOVL C00782 V=800.0 PL=0
MOVL C00783 V=800.0 PL=0
MOVL C00784 V=800.0 PL=0
MOVL C00785 V=800.0 PL=0
MOVL C00786 V=800.0 PL=0
MOVL C00787 V=800.0 PL=0
MOVL C00788 V=800.0 PL=0
MOVL C00789 V=800.0 PL=0
MOVL C00790 V=800.0 PL=0
MOVL C00791 V=800.0 PL=0
MOVL C00792 V=800.0 PL=0
MOVL C00793 V=800.0 PL=0
MOVL C00794 V=800.0 PL=0
MOVL C00795 V=800.0 PL=0
MOVL C00796 V=800.0 PL=0
MOVL C00797 V=800.0 PL=0
MOVL C00798 V=800.0 PL=0
MOVL C00799 V=800.0 PL=0
MOVL C00800 V=800.0 PL=0
MOVL C00801 V=800.0 PL=0
MOVL C00802 V=800.0 PL=0
MOVL C00803 V=800.0 PL=0
MOVL C00804 V=800.0 PL=0
MOVL C00805 V=800.0 PL=0
MOVL C00806 V=800.0 PL=0
MOVL C00807 V=800.0 PL=0
MOVL C00808 V=800.0 PL=0
MOVL C00809 V=800.0 PL=0
MOVL C00810 V=800.0 PL=0
MOVL C00811 V=800.0 PL=0
MOVL C00812 V=800.0 PL=0
MOVL C00813 V=800.0 PL=0
MOVL C00814 V=800.0 PL=0
MOVL C00815 V=800.0 PL=0
MOVL C00816 V=800.0 PL=0
MOVL C00817 V=800.0 PL=0
MOVL C00818 V=800.0 PL=0
MOVL C00819 V=800.0 PL=0
MOVL C00820 V=800.0 PL=0
MOVL C00821 V=800.0 PL=0
MOVL C00822 V=800.0 PL=0
MOVL C00823 V=800.0 PL=0
MOVL C00824 V=800.0 PL=0
MOVL C00825 V=800.0 PL=0
MOVL C00826 V=800.0 PL=0
MOVL C00827 V=800.0 PL=0
MOVL C00828 V=800.0 PL=0
MOVL C00829 V=800.0 PL=0
MOVL C00830 V=800.0 PL=0
MOVL C00831 V=800.0 PL=0
MOVL C00832 V=800.0 PL=0
MOVL C00833 V=800.0 PL=0
MOVL C00834 V=800.0 PL=0
MOVL C00835 V=800.0 PL=0
MOVL C00836 V=800.0 PL=0
MOVL C00837 V=800.0 PL=0
MOVL C00838 V=800.0 PL=0
MOVL C00839 V=800.0 PL=0
MOVL C00840 V=800.0 PL=0
MOVL C00841 V=800.0 PL=0
MOVL C00842 V=800.0 PL=0
MOVL C00843 V=800.0 PL=0
MOVL C00844 V=800.0 PL=0
MOVL C00845 V=800.0 PL=0
MOVL C00846 V=800.0 PL=0
MOVL C00847 V=800.0 PL=0
MOVL C00848 V=800.0 PL=0
MOVL C00849 V=800.0 PL=0
MOVL C00850 V=800.0 PL=0
MOVL C00851 V=800.0 PL=0
MOVL C00852 V=800.0 PL=0
MOVL C00853 V=800.0 PL=0
MOVL C00854 V=800.0 PL=0
MOVL C00855 V=800.0 PL=0
MOVL C00856 V=800.0 PL=0
MOVL C00857 V=800.0 PL=0
MOVL C00858 V=800.0 PL=0
MOVL C00859 V=800.0 PL=0
MOVL C00860 V=800.0 PL=0
MOVL C00861 V=800.0 PL=0
MOVL C00862 V=800.0 PL=0
MOVL C00863 V=800.0 PL=0
MOVL C00864 V=800.0 PL=0
MOVL C00865 V=800.0 PL=0
MOVL C00866 V=800.0 PL=0
MOVL C00867 V=800.0 PL=0
MOVL C00868 V=800.0 PL=0
MOVL C00869 V=800.0 PL=0
MOVL C00870 V=800.0 PL=0
MOVL C00871 V=800.0 PL=0
MOVL C00872 V=800.0 PL=0
MOVL C00873 V=800.0 PL=0
MOVL C00874 V=800.0 PL=0
MOVL C00875 V=800.0 PL=0
MOVL C00876 V=800.0 PL=0
MOVL C00877 V=800.0 PL=0
MOVL C00878 V=800.0 PL=0
MOVL C00879 V=800.0 PL=0
MOVL C00880 V=800.0 PL=0
MOVL C00881 V=800.0 PL=0
MOVL C00882 V=800.0 PL=0
MOVL C00883 V=800.0 PL=0
MOVL C00884 V=800.0 PL=0
MOVL C00885 V=800.0 PL=0
MOVL C00886 V=800.0 PL=0
MOVL C00887 V=800.0 PL=0
MOVL C00888 V=800.0 PL=0
MOVL C00889 V=800.0 PL=0
MOVL C00890 V=800.0 PL=0
MOVL C00891 V=800.0 PL=0
MOVL C00892 V=800.0 PL=0
MOVL C00893 V=800.0 PL=0
MOVL C00894 V=800.0 PL=0
MOVL C00895 V=800.0 PL=0
MOVL C00896 V=800.0 PL=0
MOVL C00897 V=800.0 PL=0
MOVL C00898 V=800.0 PL=0
MOVL C00899 V=800.0 PL=0
MOVL C00900 V=800.0 PL=0
MOVL C00901 V=800.0 PL=0
MOVL C00902 V=800.0 PL=0
MOVL C00903 V=800.0 PL=0
MOVL C00904 V=800.0 PL=0
MOVL C00905 V=800.0 PL=0
MOVL C00906 V=800.0 PL=0
MOVL C00907 V=800.0 PL=0
MOVL C00908 V=800.0 PL=0
MOVL C00909 V=800.0 PL=0
MOVL C00910 V=800.0 PL=0
MOVL C00911 V=800.0 PL=0
MOVL C00912 V=800.0 PL=0
MOVL C00913 V=800.0 PL=0
MOVL C00914 V=800.0 PL=0
MOVL C00915 V=800.0 PL=0
MOVL C00916 V=800.0 PL=0
MOVL C00917 V=800.0 PL=0
MOVL C00918 V=800.0 PL=0
MOVL C00919 V=800.0 PL=0
MOVL C00920 V=800.0 PL=0
MOVL C00921 V=800.0 PL=0
MOVL C00922 V=800.0 PL=0
MOVL C00923 V=800.0 PL=0
MOVL C00924 V=800.0 PL=0
MOVL C00925 V=800.0 PL=0
MOVL C00926 V=800.0 PL=0
MOVL C00927 V=800.0 PL=0
MOVL C00928 V=800.0 PL=0
MOVL C00929 V=800.0 PL=0
MOVL C00930 V=800.0 PL=0
MOVL C00931 V=800.0 PL=0
MOVL C00932 V=800.0 PL=0
MOVL C00933 V=800.0 PL=0
MOVL C00934 V=800.0 PL=0
MOVL C00935 V=800.0 PL=0
MOVL C00936 V=800.0 PL=0
MOVL C00937 V=800.0 PL=0
MOVL C00938 V=800.0 PL=0
MOVL C00939 V=800.0 PL=0
MOVL C00940 V=800.0 PL=0
MOVL C00941 V=800.0 PL=0
MOVL C00942 V=800.0 PL=0
MOVL C00943 V=800.0 PL=0
MOVL C00944 V=800.0 PL=0
MOVL C00945 V=800.0 PL=0
MOVL C00946 V=800.0 PL=0
MOVL C00947 V=800.0 PL=0
MOVL C00948 V=800.0 PL=0
MOVL C00949 V=800.0 PL=0
MOVL C00950 V=800.0 PL=0
MOVL C00951 V=800.0 PL=0
MOVL C00952 V=800.0 PL=0
MOVL C00953 V=800.0 PL=0
MOVL C00954 V=800.0 PL=0
MOVL C00955 V=800.0 PL=0
MOVL C00956 V=800.0 PL=0
MOVL C00957 V=800.0 PL=0
MOVL C00958 V=800.0 PL=0
MOVL C00959 V=800.0 PL=0
MOVL C00960 V=800.0 PL=0
MOVL C00961 V=800.0 PL=0
MOVL C00962 V=800.0 PL=0
MOVL C00963 V=800.0 PL=0
MOVL C00964 V=800.0 PL=0
MOVL C00965 V=800.0 PL=0
MOVL C00966 V=800.0 PL=0
MOVL C00967 V=800.0 PL=0
MOVL C00968 V=800.0 PL=0
MOVL C00969 V=800.0 PL=0
MOVL C00970 V=800.0 PL=0
MOVL C00971 V=800.0 PL=0
MOVL C00972 V=800.0 PL=0
MOVL C00973 V=800.0 PL=0
MOVL C00974 V=800.0 PL=0
MOVL C00975 V=800.0 PL=0
MOVL C00976 V=800.0 PL=0
MOVL C00977 V=800.0 PL=0
MOVL C00978 V=800.0 PL=0
MOVL C00979 V=800.0 PL=0
MOVL C00980 V=800.0 PL=0
MOVL C00981 V=800.0 PL=0
MOVL C00982 V=800.0 PL=0
MOVL C00983 V=800.0 PL=0
MOVL C00984 V=800.0 PL=0
MOVL C00985 V=800.0 PL=0
MOVL C00986 V=800.0 PL=0
MOVL C00987 V=800.0 PL=0
MOVL C00988 V=800.0 PL=0
MOVL C00989 V=800.0 PL=0
MOVL C00990 V=800.0 PL=0
MOVL C00991 V=800.0 PL=0
MOVL C00992 V=800.0 PL=0
MOVL C00993 V=800.0 PL=0
MOVL C00994 V=800.0 PL=0
MOVL C00995 V=800.0 PL=0
MOVL C00996 V=800.0 PL=0
MOVL C00997 V=800.0 PL=0
MOVL C00998 V=800.0 PL=0
MOVL C00999 V=800.0 PL=0
MOVL C01000 V=800.0 PL=0
MOVL C01001 V=800.0 PL=0
MOVL C01002 V=800.0 PL=0
MOVL C01003 V=800.0 PL=0
MOVL C01004 V=800.0 PL=0
MOVL C01005 V=800.0 PL=0
MOVL C01006 V=800.0 PL=0
MOVL C01007 V=800.0 PL=0
MOVL C01008 V=800.0 PL=0
MOVL C01009 V=800.0 PL=0
MOVL C01010 V=800.0 PL=0
MOVL C01011 V=800.0 PL=0
MOVL C01012 V=800.0 PL=0
MOVL C01013 V=800.0 PL=0
MOVL C01014 V=800.0 PL=0
MOVL C01015 V=800.0 PL=0
MOVL C01016 V=800.0 PL=0
MOVL C01017 V=800.0 PL=0
MOVL C01018 V=800.0 PL=0
MOVL C01019 V=800.0 PL=0
MOVL C01020 V=800.0 PL=0
MOVL C01021 V=800.0 PL=0
MOVL C01022 V=800.0 PL=0
MOVL C01023 V=800.0 PL=0
MOVL C01024 V=800.0 PL=0
MOVL C01025 V=800.0 PL=0
MOVL C01026 V=800.0 PL=0
MOVL C01027 V=800.0 PL=0
MOVL C01028 V=800.0 PL=0
MOVL C01029 V=800.0 PL=0
MOVL C01030 V=800.0 PL=0
MOVL C01031 V=800.0 PL=0
MOVL C01032 V=800.0 PL=0
MOVL C01033 V=800.0 PL=0
MOVL C01034 V=800.0 PL=0
MOVL C01035 V=800.0 PL=0
MOVL C01036 V=800.0 PL=0
MOVL C01037 V=800.0 PL=0
MOVL C01038 V=800.0 PL=0
MOVL C01039 V=800.0 PL=0
MOVL C01040 V=800.0 PL=0
MOVL C01041 V=800.0 PL=0
MOVL C01042 V=800.0 PL=0
MOVL C01043 V=800.0 PL=0
MOVL C01044 V=800.0 PL=0
MOVL C01045 V=800.0 PL=0
MOVL C01046 V=800.0 PL=0
MOVL C01047 V=800.0 PL=0
MOVL C01048 V=800.0 PL=0
MOVL C01049 V=800.0 PL=0
MOVL C01050 V=800.0 PL=0
MOVL C01051 V=800.0 PL=0
MOVL C01052 V=800.0 PL=0
MOVL C01053 V=800.0 PL=0
MOVL C01054 V=800.0 PL=0
MOVL C01055 V=800.0 PL=0
MOVL C01056 V=800.0 PL=0
MOVL C01057 V=800.0 PL=0
MOVL C01058 V=800.0 PL=0
MOVL C01059 V=800.0 PL=0
MOVL C01060 V=800.0 PL=0
MOVL C01061 V=800.0 PL=0
MOVL C01062 V=800.0 PL=0
MOVL C01063 V=800.0 PL=0
MOVL C01064 V=800.0 PL=0
MOVL C01065 V=800.0 PL=0
MOVL C01066 V=800.0 PL=0
MOVL C01067 V=800.0 PL=0
MOVL C01068 V=800.0 PL=0
MOVL C01069 V=800.0 PL=0
MOVL C01070 V=800.0 PL=0
MOVL C01071 V=800.0 PL=0
MOVL C01072 V=800.0 PL=0
MOVL C01073 V=800.0 PL=0
MOVL C01074 V=800.0 PL=0
MOVL C01075 V=800.0 PL=0
MOVL C01076 V=800.0 PL=0
MOVL C01077 V=800.0 PL=0
MOVL C01078 V=800.0 PL=0
MOVL C01079 V=800.0 PL=0
MOVL C01080 V=800.0 PL=0
MOVL C01081 V=800.0 PL=0
MOVL C01082 V=800.0 PL=0
MOVL C01083 V=800.0 PL=0
MOVL C01084 V=800.0 PL=0
MOVL C01085 V=800.0 PL=0
MOVL C01086 V=800.0 PL=0
MOVL C01087 V=800.0 PL=0
MOVL C01088 V=800.0 PL=0
MOVL C01089 V=800.0 PL=0
MOVL C01090 V=800.0 PL=0
MOVL C01091 V=800.0 PL=0
MOVL C01092 V=800.0 PL=0
MOVL C01093 V=800.0 PL=0
MOVL C01094 V=800.0 PL=0
MOVL C01095 V=800.0 PL=0
MOVL C01096 V=800.0 PL=0
MOVL C01097 V=800.0 PL=0
MOVL C01098 V=800.0 PL=0
MOVL C01099 V=800.0 PL=0
MOVL C01100 V=800.0 PL=0
MOVL C01101 V=800.0 PL=0
MOVL C01102 V=800.0 PL=0
MOVL C01103 V=800.0 PL=0
MOVL C01104 V=800.0 PL=0
MOVL C01105 V=800.0 PL=0
MOVL C01106 V=800.0 PL=0
MOVL C01107 V=800.0 PL=0
MOVL C01108 V=800.0 PL=0
MOVL C01109 V=800.0 PL=0
MOVL C01110 V=800.0 PL=0
MOVL C01111 V=800.0 PL=0
MOVL C01112 V=800.0 PL=0
MOVL C01113 V=800.0 PL=0
MOVL C01114 V=800.0 PL=0
MOVL C01115 V=800.0 PL=0
MOVL C01116 V=800.0 PL=0
MOVL C01117 V=800.0 PL=0
MOVL C01118 V=800.0 PL=0
MOVL C01119 V=800.0 PL=0
MOVL C01120 V=800.0 PL=0
MOVL C01121 V=800.0 PL=0
MOVL C01122 V=800.0 PL=0
MOVL C01123 V=800.0 PL=0
MOVL C01124 V=800.0 PL=0
MOVL C01125 V=800.0 PL=0
MOVL C01126 V=800.0 PL=0
MOVL C01127 V=800.0 PL=0
MOVL C01128 V=800.0 PL=0
MOVL C01129 V=800.0 PL=0
MOVL C01130 V=800.0 PL=0
MOVL C01131 V=800.0 PL=0
MOVL C01132 V=800.0 PL=0
MOVL C01133 V=800.0 PL=0
MOVL C01134 V=800.0 PL=0
MOVL C01135 V=800.0 PL=0
MOVL C01136 V=800.0 PL=0
MOVL C01137 V=800.0 PL=0
MOVL C01138 V=800.0 PL=0
MOVL C01139 V=800.0 PL=0
MOVL C01140 V=800.0 PL=0
MOVL C01141 V=800.0 PL=0
MOVL C01142 V=800.0 PL=0
MOVL C01143 V=800.0 PL=0
MOVL C01144 V=800.0 PL=0
MOVL C01145 V=800.0 PL=0
MOVL C01146 V=800.0 PL=0
MOVL C01147 V=800.0 PL=0
MOVL C01148 V=800.0 PL=0
MOVL C01149 V=800.0 PL=0
MOVL C01150 V=800.0 PL=0
MOVL C01151 V=800.0 PL=0
MOVL C01152 V=800.0 PL=0
MOVL C01153 V=800.0 PL=0
MOVL C01154 V=800.0 PL=0
MOVL C01155 V=800.0 PL=0
MOVL C01156 V=800.0 PL=0
MOVL C01157 V=800.0 PL=0
MOVL C01158 V=800.0 PL=0
MOVL C01159 V=800.0 PL=0
MOVL C01160 V=800.0 PL=0
MOVL C01161 V=800.0 PL=0
MOVL C01162 V=800.0 PL=0
MOVL C01163 V=800.0 PL=0
MOVL C01164 V=800.0 PL=0
MOVL C01165 V=800.0 PL=0
MOVL C01166 V=800.0 PL=0
MOVL C01167 V=800.0 PL=0
MOVL C01168 V=800.0 PL=0
MOVL C01169 V=800.0 PL=0
MOVL C01170 V=800.0 PL=0
MOVL C01171 V=800.0 PL=0
MOVL C01172 V=800.0 PL=0
MOVL C01173 V=800.0 PL=0
MOVL C01174 V=800.0 PL=0
MOVL C01175 V=800.0 PL=0
MOVL C01176 V=800.0 PL=0
MOVL C01177 V=800.0 PL=0
MOVL C01178 V=800.0 PL=0
MOVL C01179 V=800.0 PL=0
MOVL C01180 V=800.0 PL=0
MOVL C01181 V=800.0 PL=0
MOVL C01182 V=800.0 PL=0
MOVL C01183 V=800.0 PL=0
MOVL C01184 V=800.0 PL=0
MOVL C01185 V=800.0 PL=0
MOVL C01186 V=800.0 PL=0
MOVL C01187 V=800.0 PL=0
MOVL C01188 V=800.0 PL=0
MOVL C01189 V=800.0 PL=0
MOVL C01190 V=800.0 PL=0
MOVL C01191 V=800.0 PL=0
MOVL C01192 V=800.0 PL=0
MOVL C01193 V=800.0 PL=0
MOVL C01194 V=800.0 PL=0
MOVL C01195 V=800.0 PL=0
MOVL C01196 V=800.0 PL=0
MOVL C01197 V=800.0 PL=0
MOVL C01198 V=800.0 PL=0
MOVL C01199 V=800.0 PL=0
MOVL C01200 V=800.0 PL=0
MOVL C01201 V=800.0 PL=0
MOVL C01202 V=800.0 PL=0
MOVL C01203 V=800.0 PL=0
MOVL C01204 V=800.0 PL=0
MOVL C01205 V=800.0 PL=0
MOVL C01206 V=800.0 PL=0
MOVL C01207 V=800.0 PL=0
MOVL C01208 V=800.0 PL=0
MOVL C01209 V=800.0 PL=0
MOVL C01210 V=800.0 PL=0
MOVL C01211 V=800.0 PL=0
MOVL C01212 V=800.0 PL=0
MOVL C01213 V=800.0 PL=0
MOVL C01214 V=800.0 PL=0
MOVL C01215 V=800.0 PL=0
MOVL C01216 V=800.0 PL=0
MOVL C01217 V=800.0 PL=0
MOVL C01218 V=800.0 PL=0
MOVL C01219 V=800.0 PL=0
MOVL C01220 V=800.0 PL=0
MOVL C01221 V=800.0 PL=0
MOVL C01222 V=800.0 PL=0
MOVL C01223 V=800.0 PL=0
MOVL C01224 V=800.0 PL=0
MOVL C01225 V=800.0 PL=0
MOVL C01226 V=800.0 PL=0
MOVL C01227 V=800.0 PL=0
MOVL C01228 V=800.0 PL=0
MOVL C01229 V=800.0 PL=0
MOVL C01230 V=800.0 PL=0
MOVL C01231 V=800.0 PL=0
MOVL C01232 V=800.0 PL=0
MOVL C01233 V=800.0 PL=0
MOVL C01234 V=800.0 PL=0
MOVL C01235 V=800.0 PL=0
MOVL C01236 V=800.0 PL=0
MOVL C01237 V=800.0 PL=0
MOVL C01238 V=800.0 PL=0
MOVL C01239 V=800.0 PL=0
MOVL C01240 V=800.0 PL=0
MOVL C01241 V=800.0 PL=0
MOVL C01242 V=800.0 PL=0
MOVL C01243 V=800.0 PL=0
MOVL C01244 V=800.0 PL=0
MOVL C01245 V=800.0 PL=0
MOVL C01246 V=800.0 PL=0
MOVL C01247 V=800.0 PL=0
MOVL C01248 V=800.0 PL=0
MOVL C01249 V=800.0 PL=0
MOVL C01250 V=800.0 PL=0
MOVL C01251 V=800.0 PL=0
MOVL C01252 V=800.0 PL=0
MOVL C01253 V=800.0 PL=0
MOVL C01254 V=800.0 PL=0
MOVL C01255 V=800.0 PL=0
MOVL C01256 V=800.0 PL=0
MOVL C01257 V=800.0 PL=0
MOVL C01258 V=800.0 PL=0
MOVL C01259 V=800.0 PL=0
MOVL C01260 V=800.0 PL=0
MOVL C01261 V=800.0 PL=0
MOVL C01262 V=800.0 PL=0
MOVL C01263 V=800.0 PL=0
MOVL C01264 V=800.0 PL=0
MOVL C01265 V=800.0 PL=0
MOVL C01266 V=800.0 PL=0
MOVL C01267 V=800.0 PL=0
MOVL C01268 V=800.0 PL=0
MOVL C01269 V=800.0 PL=0
MOVL C01270 V=800.0 PL=0
MOVL C01271 V=800.0 PL=0
MOVL C01272 V=800.0 PL=0
MOVL C01273 V=800.0 PL=0
MOVL C01274 V=800.0 PL=0
MOVL C01275 V=800.0 PL=0
MOVL C01276 V=800.0 PL=0
MOVL C01277 V=800.0 PL=0
MOVL C01278 V=800.0 PL=0
MOVL C01279 V=800.0 PL=0
MOVL C01280 V=800.0 PL=0
MOVL C01281 V=800.0 PL=0
MOVL C01282 V=800.0 PL=0
MOVL C01283 V=800.0 PL=0
MOVL C01284 V=800.0 PL=0
MOVL C01285 V=800.0 PL=0
MOVL C01286 V=800.0 PL=0
MOVL C01287 V=800.0 PL=0
MOVL C01288 V=800.0 PL=0
MOVL C01289 V=800.0 PL=0
MOVL C01290 V=800.0 PL=0
MOVL C01291 V=800.0 PL=0
MOVL C01292 V=800.0 PL=0
MOVL C01293 V=800.0 PL=0
MOVL C01294 V=800.0 PL=0
MOVL C01295 V=800.0 PL=0
MOVL C01296 V=800.0 PL=0
MOVL C01297 V=800.0 PL=0
MOVL C01298 V=800.0 PL=0
MOVL C01299 V=800.0 PL=0
MOVL C01300 V=800.0 PL=0
MOVL C01301 V=800.0 PL=0
MOVL C01302 V=800.0 PL=0
MOVL C01303 V=800.0 PL=0
MOVL C01304 V=800.0 PL=0
MOVL C01305 V=800.0 PL=0
MOVL C01306 V=800.0 PL=0
MOVL C01307 V=800.0 PL=0
MOVL C01308 V=800.0 PL=0
MOVL C01309 V=800.0 PL=0
MOVL C01310 V=800.0 PL=0
MOVL C01311 V=800.0 PL=0
MOVL C01312 V=800.0 PL=0
MOVL C01313 V=800.0 PL=0
MOVL C01314 V=800.0 PL=0
MOVL C01315 V=800.0 PL=0
MOVL C01316 V=800.0 PL=0
MOVL C01317 V=800.0 PL=0
MOVL C01318 V=800.0 PL=0
MOVL C01319 V=800.0 PL=0
MOVL C01320 V=800.0 PL=0
MOVL C01321 V=800.0 PL=0
MOVL C01322 V=800.0 PL=0
MOVL C01323 V=800.0 PL=0
MOVL C01324 V=800.0 PL=0
MOVL C01325 V=800.0 PL=0
MOVL C01326 V=800.0 PL=0
MOVL C01327 V=800.0 PL=0
MOVL C01328 V=800.0 PL=0
MOVL C01329 V=800.0 PL=0
MOVL C01330 V=800.0 PL=0
MOVL C01331 V=800.0 PL=0
MOVL C01332 V=800.0 PL=0
MOVL C01333 V=800.0 PL=0
MOVL C01334 V=800.0 PL=0
MOVL C01335 V=800.0 PL=0
MOVL C01336 V=800.0 PL=0
MOVL C01337 V=800.0 PL=0
MOVL C01338 V=800.0 PL=0
MOVL C01339 V=800.0 PL=0
MOVL C01340 V=800.0 PL=0
MOVL C01341 V=800.0 PL=0
MOVL C01342 V=800.0 PL=0
MOVL C01343 V=800.0 PL=0
MOVL C01344 V=800.0 PL=0
MOVL C01345 V=800.0 PL=0
MOVL C01346 V=800.0 PL=0
MOVL C01347 V=800.0 PL=0
MOVL C01348 V=800.0 PL=0
MOVL C01349 V=800.0 PL=0
MOVL C01350 V=800.0 PL=0
MOVL C01351 V=800.0 PL=0
MOVL C01352 V=800.0 PL=0
MOVL C01353 V=800.0 PL=0
MOVL C01354 V=800.0 PL=0
MOVL C01355 V=800.0 PL=0
MOVL C01356 V=800.0 PL=0
MOVL C01357 V=800.0 PL=0
MOVL C01358 V=800.0 PL=0
MOVL C01359 V=800.0 PL=0
MOVL C01360 V=800.0 PL=0
MOVL C01361 V=800.0 PL=0
MOVL C01362 V=800.0 PL=0
MOVL C01363 V=800.0 PL=0
MOVL C01364 V=800.0 PL=0
MOVL C01365 V=800.0 PL=0
MOVL C01366 V=800.0 PL=0
MOVL C01367 V=800.0 PL=0
MOVL C01368 V=800.0 PL=0
MOVL C01369 V=800.0 PL=0
MOVL C01370 V=800.0 PL=0
MOVL C01371 V=800.0 PL=0
MOVL C01372 V=800.0 PL=0
MOVL C01373 V=800.0 PL=0
MOVL C01374 V=800.0 PL=0
MOVL C01375 V=800.0 PL=0
MOVL C01376 V=800.0 PL=0
MOVL C01377 V=800.0 PL=0
MOVL C01378 V=800.0 PL=0
MOVL C01379 V=800.0 PL=0
MOVL C01380 V=800.0 PL=0
MOVL C01381 V=800.0 PL=0
MOVL C01382 V=800.0 PL=0
MOVL C01383 V=800.0 PL=0
MOVL C01384 V=800.0 PL=0
MOVL C01385 V=800.0 PL=0
MOVL C01386 V=800.0 PL=0
MOVL C01387 V=800.0 PL=0
MOVL C01388 V=800.0 PL=0
MOVL C01389 V=800.0 PL=0
MOVL C01390 V=800.0 PL=0
MOVL C01391 V=800.0 PL=0
MOVL C01392 V=800.0 PL=0
MOVL C01393 V=800.0 PL=0
MOVL C01394 V=800.0 PL=0
MOVL C01395 V=800.0 PL=0
MOVL C01396 V=800.0 PL=0
MOVL C01397 V=800.0 PL=0
MOVL C01398 V=800.0 PL=0
MOVL C01399 V=800.0 PL=0
MOVL C01400 V=800.0 PL=0
MOVL C01401 V=800.0 PL=0
MOVL C01402 V=800.0 PL=0
MOVL C01403 V=800.0 PL=0
MOVL C01404 V=800.0 PL=0
MOVL C01405 V=800.0 PL=0
MOVL C01406 V=800.0 PL=0
MOVL C01407 V=800.0 PL=0
MOVL C01408 V=800.0 PL=0
MOVL C01409 V=800.0 PL=0
MOVL C01410 V=800.0 PL=0
MOVL C01411 V=800.0 PL=0
MOVL C01412 V=800.0 PL=0
MOVL C01413 V=800.0 PL=0
MOVL C01414 V=800.0 PL=0
MOVL C01415 V=800.0 PL=0
MOVL C01416 V=800.0 PL=0
MOVL C01417 V=800.0 PL=0
MOVL C01418 V=800.0 PL=0
MOVL C01419 V=800.0 PL=0
MOVL C01420 V=800.0 PL=0
MOVL C01421 V=800.0 PL=0
MOVL C01422 V=800.0 PL=0
MOVL C01423 V=800.0 PL=0
MOVL C01424 V=800.0 PL=0
MOVL C01425 V=800.0 PL=0
MOVL C01426 V=800.0 PL=0
MOVL C01427 V=800.0 PL=0
MOVL C01428 V=800.0 PL=0
MOVL C01429 V=800.0 PL=0
MOVL C01430 V=800.0 PL=0
MOVL C01431 V=800.0 PL=0
MOVL C01432 V=800.0 PL=0
MOVL C01433 V=800.0 PL=0
MOVL C01434 V=800.0 PL=0
MOVL C01435 V=800.0 PL=0
MOVL C01436 V=800.0 PL=0
MOVL C01437 V=800.0 PL=0
MOVL C01438 V=800.0 PL=0
MOVL C01439 V=800.0 PL=0
MOVL C01440 V=800.0 PL=0
MOVL C01441 V=800.0 PL=0
MOVL C01442 V=800.0 PL=0
MOVL C01443 V=800.0 PL=0
MOVL C01444 V=800.0 PL=0
MOVL C01445 V=800.0 PL=0
MOVL C01446 V=800.0 PL=0
MOVL C01447 V=800.0 PL=0
MOVL C01448 V=800.0 PL=0
MOVL C01449 V=800.0 PL=0
MOVL C01450 V=800.0 PL=0
MOVL C01451 V=800.0 PL=0
MOVL C01452 V=800.0 PL=0
MOVL C01453 V=800.0 PL=0
MOVL C01454 V=800.0 PL=0
MOVL C01455 V=800.0 PL=0
MOVL C01456 V=800.0 PL=0
MOVL C01457 V=800.0 PL=0
MOVL C01458 V=800.0 PL=0
MOVL C01459 V=800.0 PL=0
MOVL C01460 V=800.0 PL=0
MOVL C01461 V=800.0 PL=0
MOVL C01462 V=800.0 PL=0
MOVL C01463 V=800.0 PL=0
MOVL C01464 V=800.0 PL=0
MOVL C01465 V=800.0 PL=0
MOVL C01466 V=800.0 PL=0
MOVL C01467 V=800.0 PL=0
MOVL C01468 V=800.0 PL=0
MOVL C01469 V=800.0 PL=0
MOVL C01470 V=800.0 PL=0
MOVL C01471 V=800.0 PL=0
MOVL C01472 V=800.0 PL=0
MOVL C01473 V=800.0 PL=0
MOVL C01474 V=800.0 PL=0
MOVL C01475 V=800.0 PL=0
MOVL C01476 V=800.0 PL=0
MOVL C01477 V=800.0 PL=0
MOVL C01478 V=800.0 PL=0
MOVL C01479 V=800.0 PL=0
MOVL C01480 V=800.0 PL=0
MOVL C01481 V=800.0 PL=0
MOVL C01482 V=800.0 PL=0
MOVL C01483 V=800.0 PL=0
MOVL C01484 V=800.0 PL=0
MOVL C01485 V=800.0 PL=0
MOVL C01486 V=800.0 PL=0
MOVL C01487 V=800.0 PL=0
MOVL C01488 V=800.0 PL=0
MOVL C01489 V=800.0 PL=0
MOVL C01490 V=800.0 PL=0
MOVL C01491 V=800.0 PL=0
MOVL C01492 V=800.0 PL=0
MOVL C01493 V=800.0 PL=0
MOVL C01494 V=800.0 PL=0
MOVL C01495 V=800.0 PL=0
MOVL C01496 V=800.0 PL=0
MOVL C01497 V=800.0 PL=0
MOVL C01498 V=800.0 PL=0
MOVL C01499 V=800.0 PL=0
MOVL C01500 V=800.0 PL=0
MOVL C01501 V=800.0 PL=0
MOVL C01502 V=800.0 PL=0
MOVL C01503 V=800.0 PL=0
MOVL C01504 V=800.0 PL=0
MOVL C01505 V=800.0 PL=0
MOVL C01506 V=800.0 PL=0
MOVL C01507 V=800.0 PL=0
MOVL C01508 V=800.0 PL=0
MOVL C01509 V=800.0 PL=0
MOVL C01510 V=800.0 PL=0
MOVL C01511 V=800.0 PL=0
MOVL C01512 V=800.0 PL=0
MOVL C01513 V=800.0 PL=0
MOVL C01514 V=800.0 PL=0
MOVL C01515 V=800.0 PL=0
MOVL C01516 V=800.0 PL=0
MOVL C01517 V=800.0 PL=0
MOVL C01518 V=800.0 PL=0
MOVL C01519 V=800.0 PL=0
MOVL C01520 V=800.0 PL=0
MOVL C01521 V=800.0 PL=0
MOVL C01522 V=800.0 PL=0
MOVL C01523 V=800.0 PL=0
MOVL C01524 V=800.0 PL=0
MOVL C01525 V=800.0 PL=0
MOVL C01526 V=800.0 PL=0
MOVL C01527 V=800.0 PL=0
MOVL C01528 V=800.0 PL=0
MOVL C01529 V=800.0 PL=0
MOVL C01530 V=800.0 PL=0
MOVL C01531 V=800.0 PL=0
MOVL C01532 V=800.0 PL=0
MOVL C01533 V=800.0 PL=0
MOVL C01534 V=800.0 PL=0
MOVL C01535 V=800.0 PL=0
MOVL C01536 V=800.0 PL=0
MOVL C01537 V=800.0 PL=0
MOVL C01538 V=800.0 PL=0
MOVL C01539 V=800.0 PL=0
MOVL C01540 V=800.0 PL=0
MOVL C01541 V=800.0 PL=0
MOVL C01542 V=800.0 PL=0
MOVL C01543 V=800.0 PL=0
MOVL C01544 V=800.0 PL=0
MOVL C01545 V=800.0 PL=0
MOVL C01546 V=800.0 PL=0
MOVL C01547 V=800.0 PL=0
MOVL C01548 V=800.0 PL=0
MOVL C01549 V=800.0 PL=0
MOVL C01550 V=800.0 PL=0
MOVL C01551 V=800.0 PL=0
MOVL C01552 V=800.0 PL=0
MOVL C01553 V=800.0 PL=0
MOVL C01554 V=800.0 PL=0
MOVL C01555 V=800.0 PL=0
MOVL C01556 V=800.0 PL=0
MOVL C01557 V=800.0 PL=0
MOVL C01558 V=800.0 PL=0
MOVL C01559 V=800.0 PL=0
MOVL C01560 V=800.0 PL=0
MOVL C01561 V=800.0 PL=0
MOVL C01562 V=800.0 PL=0
MOVL C01563 V=800.0 PL=0
MOVL C01564 V=800.0 PL=0
MOVL C01565 V=800.0 PL=0
MOVL C01566 V=800.0 PL=0
MOVL C01567 V=800.0 PL=0
MOVL C01568 V=800.0 PL=0
MOVL C01569 V=800.0 PL=0
MOVL C01570 V=800.0 PL=0
MOVL C01571 V=800.0 PL=0
MOVL C01572 V=800.0 PL=0
MOVL C01573 V=800.0 PL=0
MOVL C01574 V=800.0 PL=0
MOVL C01575 V=800.0 PL=0
MOVL C01576 V=800.0 PL=0
MOVL C01577 V=800.0 PL=0
MOVL C01578 V=800.0 PL=0
MOVL C01579 V=800.0 PL=0
MOVL C01580 V=800.0 PL=0
MOVL C01581 V=800.0 PL=0
MOVL C01582 V=800.0 PL=0
MOVL C01583 V=800.0 PL=0
MOVL C01584 V=800.0 PL=0
MOVL C01585 V=800.0 PL=0
MOVL C01586 V=800.0 PL=0
MOVL C01587 V=800.0 PL=0
MOVL C01588 V=800.0 PL=0
MOVL C01589 V=800.0 PL=0
MOVL C01590 V=800.0 PL=0
MOVL C01591 V=800.0 PL=0
MOVL C01592 V=800.0 PL=0
MOVL C01593 V=800.0 PL=0
MOVL C01594 V=800.0 PL=0
MOVL C01595 V=800.0 PL=0
MOVL C01596 V=800.0 PL=0
MOVL C01597 V=800.0 PL=0
MOVL C01598 V=800.0 PL=0
MOVL C01599 V=800.0 PL=0
MOVL C01600 V=800.0 PL=0
MOVL C01601 V=800.0 PL=0
MOVL C01602 V=800.0 PL=0
MOVL C01603 V=800.0 PL=0
MOVL C01604 V=800.0 PL=0
MOVL C01605 V=800.0 PL=0
MOVL C01606 V=800.0 PL=0
MOVL C01607 V=800.0 PL=0
MOVL C01608 V=800.0 PL=0
MOVL C01609 V=800.0 PL=0
MOVL C01610 V=800.0 PL=0
MOVL C01611 V=800.0 PL=0
MOVL C01612 V=800.0 PL=0
MOVL C01613 V=800.0 PL=0
MOVL C01614 V=800.0 PL=0
MOVL C01615 V=800.0 PL=0
MOVL C01616 V=800.0 PL=0
MOVL C01617 V=800.0 PL=0
MOVL C01618 V=800.0 PL=0
MOVL C01619 V=800.0 PL=0
MOVL C01620 V=800.0 PL=0
MOVL C01621 V=800.0 PL=0
MOVL C01622 V=800.0 PL=0
MOVL C01623 V=800.0 PL=0
MOVL C01624 V=800.0 PL=0
MOVL C01625 V=800.0 PL=0
MOVL C01626 V=800.0 PL=0
MOVL C01627 V=800.0 PL=0
MOVL C01628 V=800.0 PL=0
MOVL C01629 V=800.0 PL=0
MOVL C01630 V=800.0 PL=0
MOVL C01631 V=800.0 PL=0
MOVL C01632 V=800.0 PL=0
MOVL C01633 V=800.0 PL=0
MOVL C01634 V=800.0 PL=0
MOVL C01635 V=800.0 PL=0
MOVL C01636 V=800.0 PL=0
MOVL C01637 V=800.0 PL=0
MOVL C01638 V=800.0 PL=0
MOVL C01639 V=800.0 PL=0
MOVL C01640 V=800.0 PL=0
MOVL C01641 V=800.0 PL=0
MOVL C01642 V=800.0 PL=0
MOVL C01643 V=800.0 PL=0
MOVL C01644 V=800.0 PL=0
MOVL C01645 V=800.0 PL=0
MOVL C01646 V=800.0 PL=0
MOVL C01647 V=800.0 PL=0
MOVL C01648 V=800.0 PL=0
MOVL C01649 V=800.0 PL=0
MOVL C01650 V=800.0 PL=0
MOVL C01651 V=800.0 PL=0
MOVL C01652 V=800.0 PL=0
MOVL C01653 V=800.0 PL=0
MOVL C01654 V=800.0 PL=0
MOVL C01655 V=800.0 PL=0
MOVL C01656 V=800.0 PL=0
MOVL C01657 V=800.0 PL=0
MOVL C01658 V=800.0 PL=0
MOVL C01659 V=800.0 PL=0
MOVL C01660 V=800.0 PL=0
MOVL C01661 V=800.0 PL=0
MOVL C01662 V=800.0 PL=0
MOVL C01663 V=800.0 PL=0
MOVL C01664 V=800.0 PL=0
MOVL C01665 V=800.0 PL=0
MOVL C01666 V=800.0 PL=0
MOVL C01667 V=800.0 PL=0
MOVL C01668 V=800.0 PL=0
MOVL C01669 V=800.0 PL=0
MOVL C01670 V=800.0 PL=0
MOVL C01671 V=800.0 PL=0
MOVL C01672 V=800.0 PL=0
MOVL C01673 V=800.0 PL=0
MOVL C01674 V=800.0 PL=0
MOVL C01675 V=800.0 PL=0
MOVL C01676 V=800.0 PL=0
MOVL C01677 V=800.0 PL=0
MOVL C01678 V=800.0 PL=0
MOVL C01679 V=800.0 PL=0
MOVL C01680 V=800.0 PL=0
MOVL C01681 V=800.0 PL=0
MOVL C01682 V=800.0 PL=0
MOVL C01683 V=800.0 PL=0
MOVL C01684 V=800.0 PL=0
MOVL C01685 V=800.0 PL=0
MOVL C01686 V=800.0 PL=0
MOVL C01687 V=800.0 PL=0
MOVL C01688 V=800.0 PL=0
MOVL C01689 V=800.0 PL=0
MOVL C01690 V=800.0 PL=0
MOVL C01691 V=800.0 PL=0
MOVL C01692 V=800.0 PL=0
MOVL C01693 V=800.0 PL=0
MOVL C01694 V=800.0 PL=0
MOVL C01695 V=800.0 PL=0
MOVL C01696 V=800.0 PL=0
MOVL C01697 V=800.0 PL=0
MOVL C01698 V=800.0 PL=0
MOVL C01699 V=800.0 PL=0
MOVL C01700 V=800.0 PL=0
MOVL C01701 V=800.0 PL=0
MOVL C01702 V=800.0 PL=0
MOVL C01703 V=800.0 PL=0
MOVL C01704 V=800.0 PL=0
MOVL C01705 V=800.0 PL=0
MOVL C01706 V=800.0 PL=0
MOVL C01707 V=800.0 PL=0
MOVL C01708 V=800.0 PL=0
MOVL C01709 V=800.0 PL=0
MOVL C01710 V=800.0 PL=0
MOVL C01711 V=800.0 PL=0
MOVL C01712 V=800.0 PL=0
MOVL C01713 V=800.0 PL=0
MOVL C01714 V=800.0 PL=0
MOVL C01715 V=800.0 PL=0
MOVL C01716 V=800.0 PL=0
MOVL C01717 V=800.0 PL=0
MOVL C01718 V=800.0 PL=0
MOVL C01719 V=800.0 PL=0
MOVL C01720 V=800.0 PL=0
MOVL C01721 V=800.0 PL=0
MOVL C01722 V=800.0 PL=0
MOVL C01723 V=800.0 PL=0
MOVL C01724 V=800.0 PL=0
MOVL C01725 V=800.0 PL=0
MOVL C01726 V=800.0 PL=0
MOVL C01727 V=800.0 PL=0
MOVL C01728 V=800.0 PL=0
MOVL C01729 V=800.0 PL=0
MOVL C01730 V=800.0 PL=0
MOVL C01731 V=800.0 PL=0
MOVL C01732 V=800.0 PL=0
MOVL C01733 V=800.0 PL=0
MOVL C01734 V=800.0 PL=0
MOVL C01735 V=800.0 PL=0
MOVL C01736 V=800.0 PL=0
MOVL C01737 V=800.0 PL=0
MOVL C01738 V=800.0 PL=0
MOVL C01739 V=800.0 PL=0
MOVL C01740 V=800.0 PL=0
MOVL C01741 V=800.0 PL=0
MOVL C01742 V=800.0 PL=0
MOVL C01743 V=800.0 PL=0
MOVL C01744 V=800.0 PL=0
MOVL C01745 V=800.0 PL=0
MOVL C01746 V=800.0 PL=0
MOVL C01747 V=800.0 PL=0
MOVL C01748 V=800.0 PL=0
MOVL C01749 V=800.0 PL=0
MOVL C01750 V=800.0 PL=0
MOVL C01751 V=800.0 PL=0
MOVL C01752 V=800.0 PL=0
MOVL C01753 V=800.0 PL=0
MOVL C01754 V=800.0 PL=0
MOVL C01755 V=800.0 PL=0
MOVL C01756 V=800.0 PL=0
MOVL C01757 V=800.0 PL=0
MOVL C01758 V=800.0 PL=0
MOVL C01759 V=800.0 PL=0
MOVL C01760 V=800.0 PL=0
MOVL C01761 V=800.0 PL=0
MOVL C01762 V=800.0 PL=0
MOVL C01763 V=800.0 PL=0
MOVL C01764 V=800.0 PL=0
MOVL C01765 V=800.0 PL=0
MOVL C01766 V=800.0 PL=0
MOVL C01767 V=800.0 PL=0
MOVL C01768 V=800.0 PL=0
MOVL C01769 V=800.0 PL=0
MOVL C01770 V=800.0 PL=0
MOVL C01771 V=800.0 PL=0
MOVL C01772 V=800.0 PL=0
MOVL C01773 V=800.0 PL=0
MOVL C01774 V=800.0 PL=0
MOVL C01775 V=800.0 PL=0
MOVL C01776 V=800.0 PL=0
MOVL C01777 V=800.0 PL=0
MOVL C01778 V=800.0 PL=0
MOVL C01779 V=800.0 PL=0
MOVL C01780 V=800.0 PL=0
MOVL C01781 V=800.0 PL=0
MOVL C01782 V=800.0 PL=0
MOVL C01783 V=800.0 PL=0
MOVL C01784 V=800.0 PL=0
MOVL C01785 V=800.0 PL=0
MOVL C01786 V=800.0 PL=0
MOVL C01787 V=800.0 PL=0
MOVL C01788 V=800.0 PL=0
MOVL C01789 V=800.0 PL=0
MOVL C01790 V=800.0 PL=0
MOVL C01791 V=800.0 PL=0
MOVL C01792 V=800.0 PL=0
MOVL C01793 V=800.0 PL=0
MOVL C01794 V=800.0 PL=0
MOVL C01795 V=800.0 PL=0
MOVL C01796 V=800.0 PL=0
MOVL C01797 V=800.0 PL=0
MOVL C01798 V=800.0 PL=0
MOVL C01799 V=800.0 PL=0
MOVL C01800 V=800.0 PL=0
MOVL C01801 V=800.0 PL=0
MOVL C01802 V=800.0 PL=0
MOVL C01803 V=800.0 PL=0
MOVL C01804 V=800.0 PL=0
MOVL C01805 V=800.0 PL=0
MOVL C01806 V=800.0 PL=0
MOVL C01807 V=800.0 PL=0
MOVL C01808 V=800.0 PL=0
MOVL C01809 V=800.0 PL=0
MOVL C01810 V=800.0 PL=0
MOVL C01811 V=800.0 PL=0
MOVL C01812 V=800.0 PL=0
MOVL C01813 V=800.0 PL=0
MOVL C01814 V=800.0 PL=0
MOVL C01815 V=800.0 PL=0
MOVL C01816 V=800.0 PL=0
MOVL C01817 V=800.0 PL=0
MOVL C01818 V=800.0 PL=0
MOVL C01819 V=800.0 PL=0
MOVL C01820 V=800.0 PL=0
MOVL C01821 V=800.0 PL=0
MOVL C01822 V=800.0 PL=0
MOVL C01823 V=800.0 PL=0
MOVL C01824 V=800.0 PL=0
MOVL C01825 V=800.0 PL=0
MOVL C01826 V=800.0 PL=0
MOVL C01827 V=800.0 PL=0
MOVL C01828 V=800.0 PL=0
MOVL C01829 V=800.0 PL=0
MOVL C01830 V=800.0 PL=0
MOVL C01831 V=800.0 PL=0
MOVL C01832 V=800.0 PL=0
MOVL C01833 V=800.0 PL=0
MOVL C01834 V=800.0 PL=0
MOVL C01835 V=800.0 PL=0
MOVL C01836 V=800.0 PL=0
MOVL C01837 V=800.0 PL=0
MOVL C01838 V=800.0 PL=0
MOVL C01839 V=800.0 PL=0
MOVL C01840 V=800.0 PL=0
MOVL C01841 V=800.0 PL=0
MOVL C01842 V=800.0 PL=0
MOVL C01843 V=800.0 PL=0
MOVL C01844 V=800.0 PL=0
MOVL C01845 V=800.0 PL=0
MOVL C01846 V=800.0 PL=0
MOVL C01847 V=800.0 PL=0
MOVL C01848 V=800.0 PL=0
MOVL C01849 V=800.0 PL=0
MOVL C01850 V=800.0 PL=0
MOVL C01851 V=800.0 PL=0
MOVL C01852 V=800.0 PL=0
MOVL C01853 V=800.0 PL=0
MOVL C01854 V=800.0 PL=0
MOVL C01855 V=800.0 PL=0
MOVL C01856 V=800.0 PL=0
MOVL C01857 V=800.0 PL=0
MOVL C01858 V=800.0 PL=0
MOVL C01859 V=800.0 PL=0
MOVL C01860 V=800.0 PL=0
MOVL C01861 V=800.0 PL=0
MOVL C01862 V=800.0 PL=0
MOVL C01863 V=800.0 PL=0
MOVL C01864 V=800.0 PL=0
MOVL C01865 V=800.0 PL=0
MOVL C01866 V=800.0 PL=0
MOVL C01867 V=800.0 PL=0
MOVL C01868 V=800.0 PL=0
MOVL C01869 V=800.0 PL=0
MOVL C01870 V=800.0 PL=0
MOVL C01871 V=800.0 PL=0
MOVL C01872 V=800.0 PL=0
MOVL C01873 V=800.0 PL=0
MOVL C01874 V=800.0 PL=0
MOVL C01875 V=800.0 PL=0
MOVL C01876 V=800.0 PL=0
MOVL C01877 V=800.0 PL=0
MOVL C01878 V=800.0 PL=0
MOVL C01879 V=800.0 PL=0
MOVL C01880 V=800.0 PL=0
MOVL C01881 V=800.0 PL=0
MOVL C01882 V=800.0 PL=0
MOVL C01883 V=800.0 PL=0
MOVL C01884 V=800.0 PL=0
MOVL C01885 V=800.0 PL=0
MOVL C01886 V=800.0 PL=0
MOVL C01887 V=800.0 PL=0
MOVL C01888 V=800.0 PL=0
MOVL C01889 V=800.0 PL=0
MOVL C01890 V=800.0 PL=0
MOVL C01891 V=800.0 PL=0
MOVL C01892 V=800.0 PL=0
MOVL C01893 V=800.0 PL=0
MOVL C01894 V=800.0 PL=0
MOVL C01895 V=800.0 PL=0
MOVL C01896 V=800.0 PL=0
MOVL C01897 V=800.0 PL=0
MOVL C01898 V=800.0 PL=0
MOVL C01899 V=800.0 PL=0
MOVL C01900 V=800.0 PL=0
MOVL C01901 V=800.0 PL=0
MOVL C01902 V=800.0 PL=0
MOVL C01903 V=800.0 PL=0
MOVL C01904 V=800.0 PL=0
MOVL C01905 V=800.0 PL=0
MOVL C01906 V=800.0 PL=0
MOVL C01907 V=800.0 PL=0
MOVL C01908 V=800.0 PL=0
MOVL C01909 V=800.0 PL=0
MOVL C01910 V=800.0 PL=0
MOVL C01911 V=800.0 PL=0
MOVL C01912 V=800.0 PL=0
MOVL C01913 V=800.0 PL=0
MOVL C01914 V=800.0 PL=0
MOVL C01915 V=800.0 PL=0
MOVL C01916 V=800.0 PL=0
MOVL C01917 V=800.0 PL=0
MOVL C01918 V=800.0 PL=0
MOVL C01919 V=800.0 PL=0
MOVL C01920 V=800.0 PL=0
MOVL C01921 V=800.0 PL=0
MOVL C01922 V=800.0 PL=0
MOVL C01923 V=800.0 PL=0
MOVL C01924 V=800.0 PL=0
MOVL C01925 V=800.0 PL=0
MOVL C01926 V=800.0 PL=0
MOVL C01927 V=800.0 PL=0
MOVL C01928 V=800.0 PL=0
MOVL C01929 V=800.0 PL=0
MOVL C01930 V=800.0 PL=0
MOVL C01931 V=800.0 PL=0
MOVL C01932 V=800.0 PL=0
MOVL C01933 V=800.0 PL=0
MOVL C01934 V=800.0 PL=0
MOVL C01935 V=800.0 PL=0
MOVL C01936 V=800.0 PL=0
MOVL C01937 V=800.0 PL=0
MOVL C01938 V=800.0 PL=0
MOVL C01939 V=800.0 PL=0
MOVL C01940 V=800.0 PL=0
MOVL C01941 V=800.0 PL=0
MOVL C01942 V=800.0 PL=0
MOVL C01943 V=800.0 PL=0
MOVL C01944 V=800.0 PL=0
MOVL C01945 V=800.0 PL=0
MOVL C01946 V=800.0 PL=0
MOVL C01947 V=800.0 PL=0
MOVL C01948 V=800.0 PL=0
MOVL C01949 V=800.0 PL=0
MOVL C01950 V=800.0 PL=0
MOVL C01951 V=800.0 PL=0
MOVL C01952 V=800.0 PL=0
MOVL C01953 V=800.0 PL=0
MOVL C01954 V=800.0 PL=0
MOVL C01955 V=800.0 PL=0
MOVL C01956 V=800.0 PL=0
MOVL C01957 V=800.0 PL=0
MOVL C01958 V=800.0 PL=0
MOVL C01959 V=800.0 PL=0
MOVL C01960 V=800.0 PL=0
MOVL C01961 V=800.0 PL=0
MOVL C01962 V=800.0 PL=0
MOVL C01963 V=800.0 PL=0
MOVL C01964 V=800.0 PL=0
MOVL C01965 V=800.0 PL=0
MOVL C01966 V=800.0 PL=0
MOVL C01967 V=800.0 PL=0
MOVL C01968 V=800.0 PL=0
MOVL C01969 V=800.0 PL=0
MOVL C01970 V=800.0 PL=0
MOVL C01971 V=800.0 PL=0
MOVL C01972 V=800.0 PL=0
MOVL C01973 V=800.0 PL=0
MOVL C01974 V=800.0 PL=0
MOVL C01975 V=800.0 PL=0
MOVL C01976 V=800.0 PL=0
MOVL C01977 V=800.0 PL=0
MOVL C01978 V=800.0 PL=0
MOVL C01979 V=800.0 PL=0
MOVL C01980 V=800.0 PL=0
MOVL C01981 V=800.0 PL=0
MOVL C01982 V=800.0 PL=0
